REGION Network 13: MB3 Code 3034 - Rotazione Ribalta -AX_POS
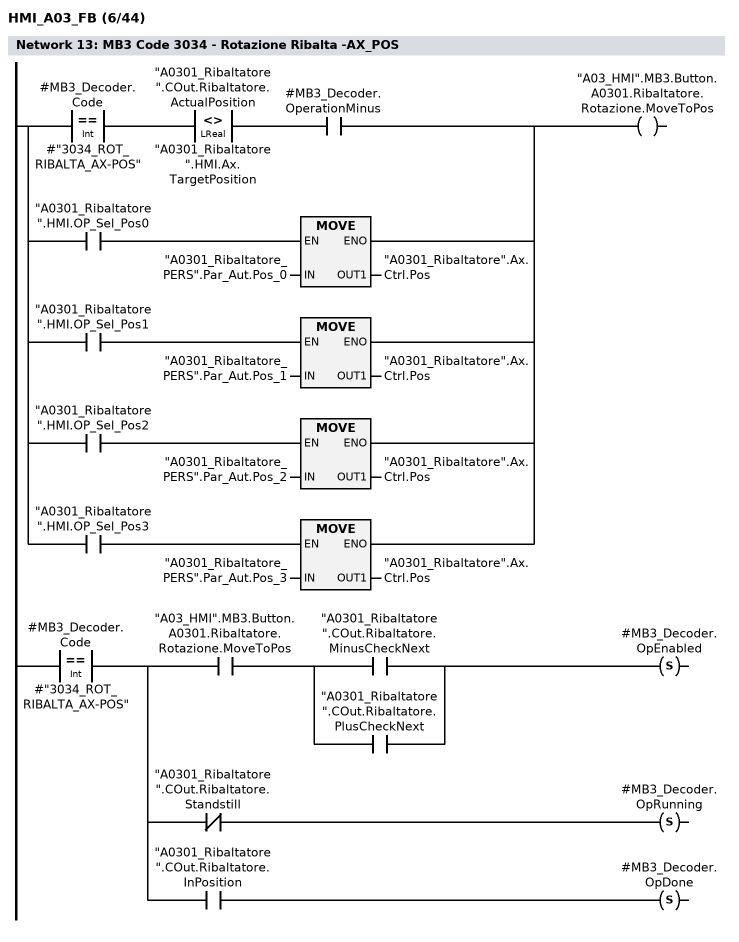
   RUNG wire#powerrail
      { S7_Templates := "SrcType := Int" } EQ_Contact(in1 := #MB3_Decoder.Code, in2 := #"3034_ROT_RIBALTA_AX-POS")
      { S7_Templates := "SrcType := LReal" } NE_Contact(in1 := "A0301_Ribaltatore".COut.Ribaltatore.ActualPosition, in2 := "A0301_Ribaltatore".HMI.Ax.TargetPosition)
      Contact( #MB3_Decoder.OperationMinus )
      wire#w1
      Coil( "A03_HMI".MB3.Button.A0301.Ribaltatore.Rotazione.MoveToPos )
   END_RUNG
   RUNG wire#powerrail
      Contact( "A0301_Ribaltatore".HMI.OP_Sel_Pos0 )
      Move(in := "A0301_Ribaltatore_PERS".Par_Aut.Pos_0, out1 => "A0301_Ribaltatore".Ax.Ctrl.Pos)
   END_RUNG wire#w1
   RUNG wire#powerrail
      Contact( "A0301_Ribaltatore".HMI.OP_Sel_Pos1 )
      Move(in := "A0301_Ribaltatore_PERS".Par_Aut.Pos_1, out1 => "A0301_Ribaltatore".Ax.Ctrl.Pos)
   END_RUNG wire#w1
   RUNG wire#powerrail
      Contact( "A0301_Ribaltatore".HMI.OP_Sel_Pos2 )
      Move(in := "A0301_Ribaltatore_PERS".Par_Aut.Pos_2, out1 => "A0301_Ribaltatore".Ax.Ctrl.Pos)
   END_RUNG wire#w1
   RUNG wire#powerrail
      Contact( "A0301_Ribaltatore".HMI.OP_Sel_Pos3 )
      Move(in := "A0301_Ribaltatore_PERS".Par_Aut.Pos_3, out1 => "A0301_Ribaltatore".Ax.Ctrl.Pos)
   END_RUNG wire#w1
   RUNG wire#powerrail
      { S7_Templates := "SrcType := Int" } EQ_Contact(in1 := #MB3_Decoder.Code, in2 := #"3034_ROT_RIBALTA_AX-POS")
      wire#w2
      Contact( "A03_HMI".MB3.Button.A0301.Ribaltatore.Rotazione.MoveToPos )
      wire#w3
      Contact( "A0301_Ribaltatore".COut.Ribaltatore.MinusCheckNext )
      wire#w4
      S_Coil( #MB3_Decoder.OpEnabled )
   END_RUNG
   RUNG wire#w3
      Contact( "A0301_Ribaltatore".COut.Ribaltatore.PlusCheckNext )
   END_RUNG wire#w4
   RUNG wire#w2
      I_Contact( "A0301_Ribaltatore".COut.Ribaltatore.Standstill )
      S_Coil( #MB3_Decoder.OpRunning )
   END_RUNG
   RUNG wire#w2
      Contact( "A0301_Ribaltatore".COut.Ribaltatore.InPosition )
      S_Coil( #MB3_Decoder.OpDone )
   END_RUNG
   // the same network as SCL:
   IF "A0301_Ribaltatore".HMI.OP_Sel_Pos0 THEN
       "A0301_Ribaltatore".Ax.Ctrl.Pos := "A0301_Ribaltatore_PERS".Par_Aut.Pos_0;
   END_IF;
   IF "A0301_Ribaltatore".HMI.OP_Sel_Pos1 THEN
       "A0301_Ribaltatore".Ax.Ctrl.Pos := "A0301_Ribaltatore_PERS".Par_Aut.Pos_1;
   END_IF;
   IF "A0301_Ribaltatore".HMI.OP_Sel_Pos2 THEN
       "A0301_Ribaltatore".Ax.Ctrl.Pos := "A0301_Ribaltatore_PERS".Par_Aut.Pos_2;
   END_IF;
   IF "A0301_Ribaltatore".HMI.OP_Sel_Pos3 THEN
       "A0301_Ribaltatore".Ax.Ctrl.Pos := "A0301_Ribaltatore_PERS".Par_Aut.Pos_3;
   END_IF;
   "A03_HMI".MB3.Button.A0301.Ribaltatore.Rotazione.MoveToPos := ((#MB3_Decoder.Code = #"3034_ROT_RIBALTA_AX-POS") AND ("A0301_Ribaltatore".COut.Ribaltatore.ActualPosition <> "A0301_Ribaltatore".HMI.Ax.TargetPosition) AND #MB3_Decoder.OperationMinus) OR "A0301_Ribaltatore".HMI.OP_Sel_Pos0 OR "A0301_Ribaltatore".HMI.OP_Sel_Pos1 OR "A0301_Ribaltatore".HMI.OP_Sel_Pos2 OR "A0301_Ribaltatore".HMI.OP_Sel_Pos3;
   #_w1 := #MB3_Decoder.Code = #"3034_ROT_RIBALTA_AX-POS";
   IF #_w1 AND "A03_HMI".MB3.Button.A0301.Ribaltatore.Rotazione.MoveToPos AND ("A0301_Ribaltatore".COut.Ribaltatore.MinusCheckNext OR "A0301_Ribaltatore".COut.Ribaltatore.PlusCheckNext) THEN
       #MB3_Decoder.OpEnabled := TRUE;
   END_IF;
   IF #_w1 AND NOT "A0301_Ribaltatore".COut.Ribaltatore.Standstill THEN
       #MB3_Decoder.OpRunning := TRUE;
   END_IF;
   IF #_w1 AND "A0301_Ribaltatore".COut.Ribaltatore.InPosition THEN #MB3_Decoder.OpDone := TRUE; END_IF;
END_REGION

REGION Network 14: MB3 Code 6008 - Rotazione Ribalta - OP POS0
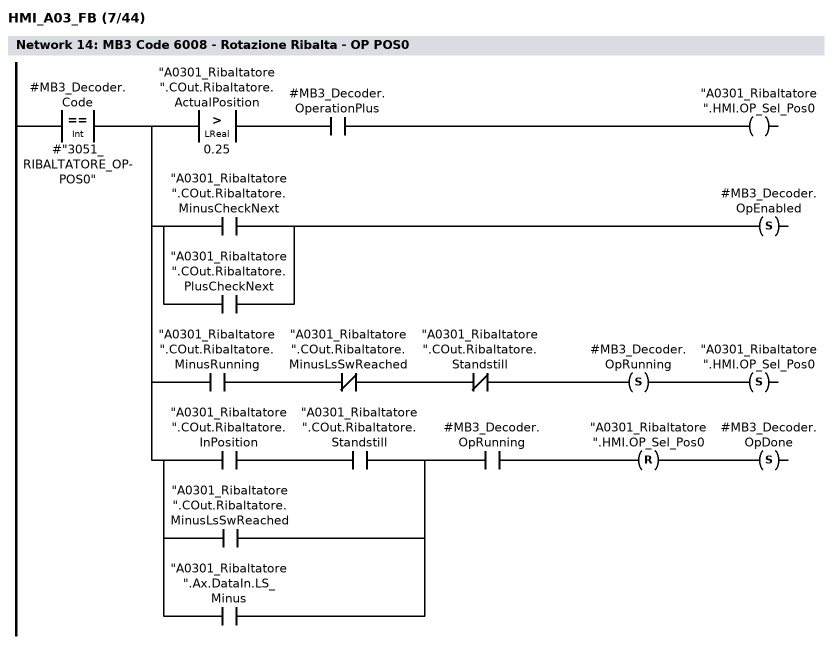
   RUNG wire#powerrail
      { S7_Templates := "SrcType := Int" } EQ_Contact(in1 := #MB3_Decoder.Code, in2 := #"3051_RIBALTATORE_OP-POS0")
      wire#w1
      { S7_Templates := "SrcType := LReal" } GT_Contact(in1 := "A0301_Ribaltatore".COut.Ribaltatore.ActualPosition, in2 := 0.25)
      Contact( #MB3_Decoder.OperationPlus )
      Coil( "A0301_Ribaltatore".HMI.OP_Sel_Pos0 )
   END_RUNG
   RUNG wire#w1
      Contact( "A0301_Ribaltatore".COut.Ribaltatore.MinusCheckNext )
      wire#w2
      S_Coil( #MB3_Decoder.OpEnabled )
   END_RUNG
   RUNG wire#w1
      Contact( "A0301_Ribaltatore".COut.Ribaltatore.PlusCheckNext )
   END_RUNG wire#w2
   RUNG wire#w1
      Contact( "A0301_Ribaltatore".COut.Ribaltatore.MinusRunning )
      I_Contact( "A0301_Ribaltatore".COut.Ribaltatore.MinusLsSwReached )
      I_Contact( "A0301_Ribaltatore".COut.Ribaltatore.Standstill )
      S_Coil( #MB3_Decoder.OpRunning )
      S_Coil( "A0301_Ribaltatore".HMI.OP_Sel_Pos0 )
   END_RUNG
   RUNG wire#w1
      Contact( "A0301_Ribaltatore".COut.Ribaltatore.InPosition )
      Contact( "A0301_Ribaltatore".COut.Ribaltatore.Standstill )
      wire#w3
      Contact( #MB3_Decoder.OpRunning )
      R_Coil( "A0301_Ribaltatore".HMI.OP_Sel_Pos0 )
      S_Coil( #MB3_Decoder.OpDone )
   END_RUNG
   RUNG wire#w1
      Contact( "A0301_Ribaltatore".COut.Ribaltatore.MinusLsSwReached )
   END_RUNG wire#w3
   RUNG wire#w1
      Contact( "A0301_Ribaltatore".Ax.DataIn.LS_Minus )
   END_RUNG wire#w3
   // the same network as SCL:
   #_w1 := #MB3_Decoder.Code = #"3051_RIBALTATORE_OP-POS0";
   "A0301_Ribaltatore".HMI.OP_Sel_Pos0 := #_w1 AND ("A0301_Ribaltatore".COut.Ribaltatore.ActualPosition > 0.25) AND #MB3_Decoder.OperationPlus;
   IF #_w1 AND ("A0301_Ribaltatore".COut.Ribaltatore.MinusCheckNext OR "A0301_Ribaltatore".COut.Ribaltatore.PlusCheckNext) THEN
       #MB3_Decoder.OpEnabled := TRUE;
   END_IF;
   IF #_w1 AND "A0301_Ribaltatore".COut.Ribaltatore.MinusRunning AND NOT "A0301_Ribaltatore".COut.Ribaltatore.MinusLsSwReached AND NOT "A0301_Ribaltatore".COut.Ribaltatore.Standstill THEN
       #MB3_Decoder.OpRunning := TRUE;
       "A0301_Ribaltatore".HMI.OP_Sel_Pos0 := TRUE;
   END_IF;
   IF #_w1 AND (("A0301_Ribaltatore".COut.Ribaltatore.InPosition AND "A0301_Ribaltatore".COut.Ribaltatore.Standstill) OR "A0301_Ribaltatore".COut.Ribaltatore.MinusLsSwReached OR "A0301_Ribaltatore".Ax.DataIn.LS_Minus) AND #MB3_Decoder.OpRunning THEN
       "A0301_Ribaltatore".HMI.OP_Sel_Pos0 := FALSE;
       #MB3_Decoder.OpDone := TRUE;
   END_IF;
END_REGION

REGION Network 15: MB3 Code 6009 - Rotazione Ribalta - OP POS1
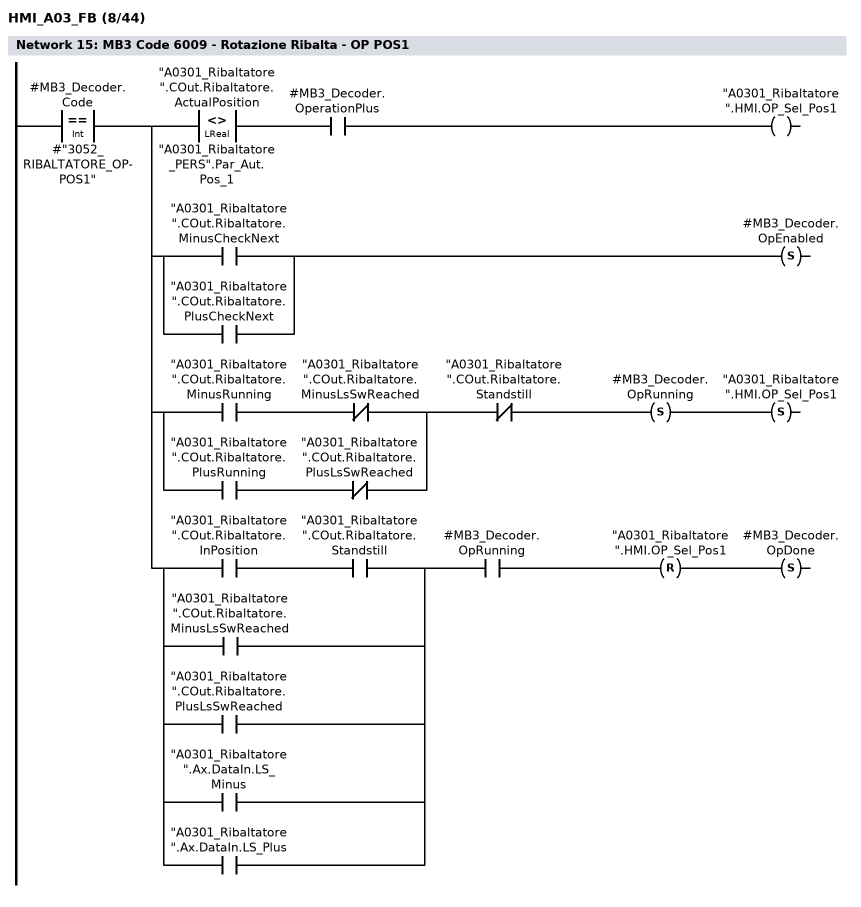
   RUNG wire#powerrail
      { S7_Templates := "SrcType := Int" } EQ_Contact(in1 := #MB3_Decoder.Code, in2 := #"3052_RIBALTATORE_OP-POS1")
      wire#w1
      { S7_Templates := "SrcType := LReal" } NE_Contact(in1 := "A0301_Ribaltatore".COut.Ribaltatore.ActualPosition, in2 := "A0301_Ribaltatore_PERS".Par_Aut.Pos_1)
      Contact( #MB3_Decoder.OperationPlus )
      Coil( "A0301_Ribaltatore".HMI.OP_Sel_Pos1 )
   END_RUNG
   RUNG wire#w1
      Contact( "A0301_Ribaltatore".COut.Ribaltatore.MinusCheckNext )
      wire#w2
      S_Coil( #MB3_Decoder.OpEnabled )
   END_RUNG
   RUNG wire#w1
      Contact( "A0301_Ribaltatore".COut.Ribaltatore.PlusCheckNext )
   END_RUNG wire#w2
   RUNG wire#w1
      Contact( "A0301_Ribaltatore".COut.Ribaltatore.MinusRunning )
      I_Contact( "A0301_Ribaltatore".COut.Ribaltatore.MinusLsSwReached )
      wire#w3
      I_Contact( "A0301_Ribaltatore".COut.Ribaltatore.Standstill )
      S_Coil( #MB3_Decoder.OpRunning )
      S_Coil( "A0301_Ribaltatore".HMI.OP_Sel_Pos1 )
   END_RUNG
   RUNG wire#w1
      Contact( "A0301_Ribaltatore".COut.Ribaltatore.PlusRunning )
      I_Contact( "A0301_Ribaltatore".COut.Ribaltatore.PlusLsSwReached )
   END_RUNG wire#w3
   RUNG wire#w1
      Contact( "A0301_Ribaltatore".COut.Ribaltatore.InPosition )
      Contact( "A0301_Ribaltatore".COut.Ribaltatore.Standstill )
      wire#w4
      Contact( #MB3_Decoder.OpRunning )
      R_Coil( "A0301_Ribaltatore".HMI.OP_Sel_Pos1 )
      S_Coil( #MB3_Decoder.OpDone )
   END_RUNG
   RUNG wire#w1
      Contact( "A0301_Ribaltatore".COut.Ribaltatore.MinusLsSwReached )
   END_RUNG wire#w4
   RUNG wire#w1
      Contact( "A0301_Ribaltatore".COut.Ribaltatore.PlusLsSwReached )
   END_RUNG wire#w4
   RUNG wire#w1
      Contact( "A0301_Ribaltatore".Ax.DataIn.LS_Minus )
   END_RUNG wire#w4
   RUNG wire#w1
      Contact( "A0301_Ribaltatore".Ax.DataIn.LS_Plus )
   END_RUNG wire#w4
   // the same network as SCL:
   #_w1 := #MB3_Decoder.Code = #"3052_RIBALTATORE_OP-POS1";
   "A0301_Ribaltatore".HMI.OP_Sel_Pos1 := #_w1 AND ("A0301_Ribaltatore".COut.Ribaltatore.ActualPosition <> "A0301_Ribaltatore_PERS".Par_Aut.Pos_1) AND #MB3_Decoder.OperationPlus;
   IF #_w1 AND ("A0301_Ribaltatore".COut.Ribaltatore.MinusCheckNext OR "A0301_Ribaltatore".COut.Ribaltatore.PlusCheckNext) THEN
       #MB3_Decoder.OpEnabled := TRUE;
   END_IF;
   IF #_w1 AND (("A0301_Ribaltatore".COut.Ribaltatore.MinusRunning AND NOT "A0301_Ribaltatore".COut.Ribaltatore.MinusLsSwReached) OR ("A0301_Ribaltatore".COut.Ribaltatore.PlusRunning AND NOT "A0301_Ribaltatore".COut.Ribaltatore.PlusLsSwReached)) AND NOT "A0301_Ribaltatore".COut.Ribaltatore.Standstill THEN
       #MB3_Decoder.OpRunning := TRUE;
       "A0301_Ribaltatore".HMI.OP_Sel_Pos1 := TRUE;
   END_IF;
   IF #_w1 AND (("A0301_Ribaltatore".COut.Ribaltatore.InPosition AND "A0301_Ribaltatore".COut.Ribaltatore.Standstill) OR "A0301_Ribaltatore".COut.Ribaltatore.MinusLsSwReached OR "A0301_Ribaltatore".COut.Ribaltatore.PlusLsSwReached OR "A0301_Ribaltatore".Ax.DataIn.LS_Minus OR "A0301_Ribaltatore".Ax.DataIn.LS_Plus) AND #MB3_Decoder.OpRunning THEN
       "A0301_Ribaltatore".HMI.OP_Sel_Pos1 := FALSE;
       #MB3_Decoder.OpDone := TRUE;
   END_IF;
END_REGION

REGION Network 16: MB3 Code 6010 - Rotazione Ribalta - OP POS2
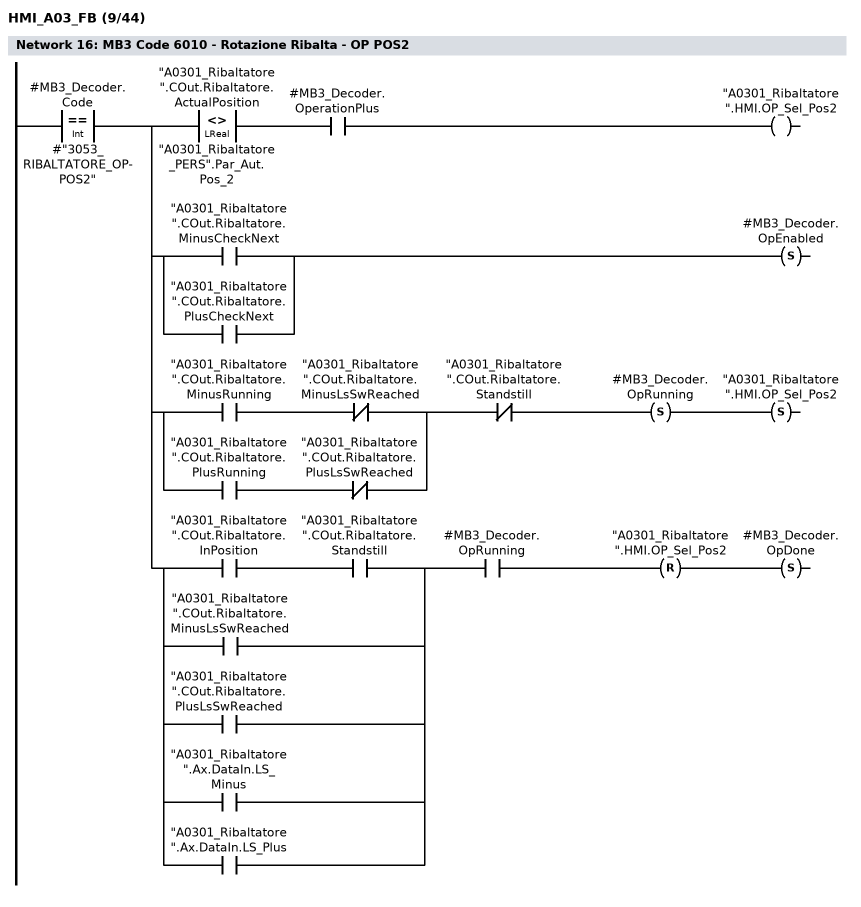
   RUNG wire#powerrail
      { S7_Templates := "SrcType := Int" } EQ_Contact(in1 := #MB3_Decoder.Code, in2 := #"3053_RIBALTATORE_OP-POS2")
      wire#w1
      { S7_Templates := "SrcType := LReal" } NE_Contact(in1 := "A0301_Ribaltatore".COut.Ribaltatore.ActualPosition, in2 := "A0301_Ribaltatore_PERS".Par_Aut.Pos_2)
      Contact( #MB3_Decoder.OperationPlus )
      Coil( "A0301_Ribaltatore".HMI.OP_Sel_Pos2 )
   END_RUNG
   RUNG wire#w1
      Contact( "A0301_Ribaltatore".COut.Ribaltatore.MinusCheckNext )
      wire#w2
      S_Coil( #MB3_Decoder.OpEnabled )
   END_RUNG
   RUNG wire#w1
      Contact( "A0301_Ribaltatore".COut.Ribaltatore.PlusCheckNext )
   END_RUNG wire#w2
   RUNG wire#w1
      Contact( "A0301_Ribaltatore".COut.Ribaltatore.MinusRunning )
      I_Contact( "A0301_Ribaltatore".COut.Ribaltatore.MinusLsSwReached )
      wire#w3
      I_Contact( "A0301_Ribaltatore".COut.Ribaltatore.Standstill )
      S_Coil( #MB3_Decoder.OpRunning )
      S_Coil( "A0301_Ribaltatore".HMI.OP_Sel_Pos2 )
   END_RUNG
   RUNG wire#w1
      Contact( "A0301_Ribaltatore".COut.Ribaltatore.PlusRunning )
      I_Contact( "A0301_Ribaltatore".COut.Ribaltatore.PlusLsSwReached )
   END_RUNG wire#w3
   RUNG wire#w1
      Contact( "A0301_Ribaltatore".COut.Ribaltatore.InPosition )
      Contact( "A0301_Ribaltatore".COut.Ribaltatore.Standstill )
      wire#w4
      Contact( #MB3_Decoder.OpRunning )
      R_Coil( "A0301_Ribaltatore".HMI.OP_Sel_Pos2 )
      S_Coil( #MB3_Decoder.OpDone )
   END_RUNG
   RUNG wire#w1
      Contact( "A0301_Ribaltatore".COut.Ribaltatore.MinusLsSwReached )
   END_RUNG wire#w4
   RUNG wire#w1
      Contact( "A0301_Ribaltatore".COut.Ribaltatore.PlusLsSwReached )
   END_RUNG wire#w4
   RUNG wire#w1
      Contact( "A0301_Ribaltatore".Ax.DataIn.LS_Minus )
   END_RUNG wire#w4
   RUNG wire#w1
      Contact( "A0301_Ribaltatore".Ax.DataIn.LS_Plus )
   END_RUNG wire#w4
   // the same network as SCL:
   #_w1 := #MB3_Decoder.Code = #"3053_RIBALTATORE_OP-POS2";
   "A0301_Ribaltatore".HMI.OP_Sel_Pos2 := #_w1 AND ("A0301_Ribaltatore".COut.Ribaltatore.ActualPosition <> "A0301_Ribaltatore_PERS".Par_Aut.Pos_2) AND #MB3_Decoder.OperationPlus;
   IF #_w1 AND ("A0301_Ribaltatore".COut.Ribaltatore.MinusCheckNext OR "A0301_Ribaltatore".COut.Ribaltatore.PlusCheckNext) THEN
       #MB3_Decoder.OpEnabled := TRUE;
   END_IF;
   IF #_w1 AND (("A0301_Ribaltatore".COut.Ribaltatore.MinusRunning AND NOT "A0301_Ribaltatore".COut.Ribaltatore.MinusLsSwReached) OR ("A0301_Ribaltatore".COut.Ribaltatore.PlusRunning AND NOT "A0301_Ribaltatore".COut.Ribaltatore.PlusLsSwReached)) AND NOT "A0301_Ribaltatore".COut.Ribaltatore.Standstill THEN
       #MB3_Decoder.OpRunning := TRUE;
       "A0301_Ribaltatore".HMI.OP_Sel_Pos2 := TRUE;
   END_IF;
   IF #_w1 AND (("A0301_Ribaltatore".COut.Ribaltatore.InPosition AND "A0301_Ribaltatore".COut.Ribaltatore.Standstill) OR "A0301_Ribaltatore".COut.Ribaltatore.MinusLsSwReached OR "A0301_Ribaltatore".COut.Ribaltatore.PlusLsSwReached OR "A0301_Ribaltatore".Ax.DataIn.LS_Minus OR "A0301_Ribaltatore".Ax.DataIn.LS_Plus) AND #MB3_Decoder.OpRunning THEN
       "A0301_Ribaltatore".HMI.OP_Sel_Pos2 := FALSE;
       #MB3_Decoder.OpDone := TRUE;
   END_IF;
END_REGION

REGION Network 17: MB3 Code 6011 - Rotazione Ribalta - OP POS3
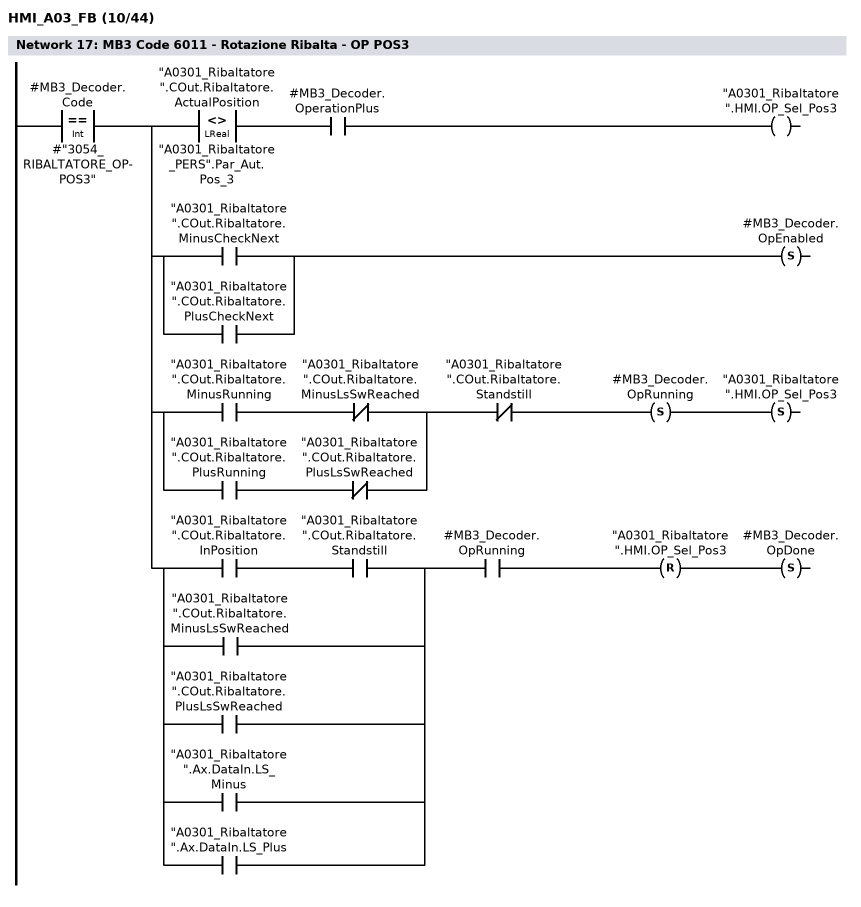
   RUNG wire#powerrail
      { S7_Templates := "SrcType := Int" } EQ_Contact(in1 := #MB3_Decoder.Code, in2 := #"3054_RIBALTATORE_OP-POS3")
      wire#w1
      { S7_Templates := "SrcType := LReal" } NE_Contact(in1 := "A0301_Ribaltatore".COut.Ribaltatore.ActualPosition, in2 := "A0301_Ribaltatore_PERS".Par_Aut.Pos_3)
      Contact( #MB3_Decoder.OperationPlus )
      Coil( "A0301_Ribaltatore".HMI.OP_Sel_Pos3 )
   END_RUNG
   RUNG wire#w1
      Contact( "A0301_Ribaltatore".COut.Ribaltatore.MinusCheckNext )
      wire#w2
      S_Coil( #MB3_Decoder.OpEnabled )
   END_RUNG
   RUNG wire#w1
      Contact( "A0301_Ribaltatore".COut.Ribaltatore.PlusCheckNext )
   END_RUNG wire#w2
   RUNG wire#w1
      Contact( "A0301_Ribaltatore".COut.Ribaltatore.MinusRunning )
      I_Contact( "A0301_Ribaltatore".COut.Ribaltatore.MinusLsSwReached )
      wire#w3
      I_Contact( "A0301_Ribaltatore".COut.Ribaltatore.Standstill )
      S_Coil( #MB3_Decoder.OpRunning )
      S_Coil( "A0301_Ribaltatore".HMI.OP_Sel_Pos3 )
   END_RUNG
   RUNG wire#w1
      Contact( "A0301_Ribaltatore".COut.Ribaltatore.PlusRunning )
      I_Contact( "A0301_Ribaltatore".COut.Ribaltatore.PlusLsSwReached )
   END_RUNG wire#w3
   RUNG wire#w1
      Contact( "A0301_Ribaltatore".COut.Ribaltatore.InPosition )
      Contact( "A0301_Ribaltatore".COut.Ribaltatore.Standstill )
      wire#w4
      Contact( #MB3_Decoder.OpRunning )
      R_Coil( "A0301_Ribaltatore".HMI.OP_Sel_Pos3 )
      S_Coil( #MB3_Decoder.OpDone )
   END_RUNG
   RUNG wire#w1
      Contact( "A0301_Ribaltatore".COut.Ribaltatore.MinusLsSwReached )
   END_RUNG wire#w4
   RUNG wire#w1
      Contact( "A0301_Ribaltatore".COut.Ribaltatore.PlusLsSwReached )
   END_RUNG wire#w4
   RUNG wire#w1
      Contact( "A0301_Ribaltatore".Ax.DataIn.LS_Minus )
   END_RUNG wire#w4
   RUNG wire#w1
      Contact( "A0301_Ribaltatore".Ax.DataIn.LS_Plus )
   END_RUNG wire#w4
   // the same network as SCL:
   #_w1 := #MB3_Decoder.Code = #"3054_RIBALTATORE_OP-POS3";
   "A0301_Ribaltatore".HMI.OP_Sel_Pos3 := #_w1 AND ("A0301_Ribaltatore".COut.Ribaltatore.ActualPosition <> "A0301_Ribaltatore_PERS".Par_Aut.Pos_3) AND #MB3_Decoder.OperationPlus;
   IF #_w1 AND ("A0301_Ribaltatore".COut.Ribaltatore.MinusCheckNext OR "A0301_Ribaltatore".COut.Ribaltatore.PlusCheckNext) THEN
       #MB3_Decoder.OpEnabled := TRUE;
   END_IF;
   IF #_w1 AND (("A0301_Ribaltatore".COut.Ribaltatore.MinusRunning AND NOT "A0301_Ribaltatore".COut.Ribaltatore.MinusLsSwReached) OR ("A0301_Ribaltatore".COut.Ribaltatore.PlusRunning AND NOT "A0301_Ribaltatore".COut.Ribaltatore.PlusLsSwReached)) AND NOT "A0301_Ribaltatore".COut.Ribaltatore.Standstill THEN
       #MB3_Decoder.OpRunning := TRUE;
       "A0301_Ribaltatore".HMI.OP_Sel_Pos3 := TRUE;
   END_IF;
   IF #_w1 AND (("A0301_Ribaltatore".COut.Ribaltatore.InPosition AND "A0301_Ribaltatore".COut.Ribaltatore.Standstill) OR "A0301_Ribaltatore".COut.Ribaltatore.MinusLsSwReached OR "A0301_Ribaltatore".COut.Ribaltatore.PlusLsSwReached OR "A0301_Ribaltatore".Ax.DataIn.LS_Minus OR "A0301_Ribaltatore".Ax.DataIn.LS_Plus) AND #MB3_Decoder.OpRunning THEN
       "A0301_Ribaltatore".HMI.OP_Sel_Pos3 := FALSE;
       #MB3_Decoder.OpDone := TRUE;
   END_IF;
END_REGION

REGION Network 18: MB3 Code 3041 - Fermi P4
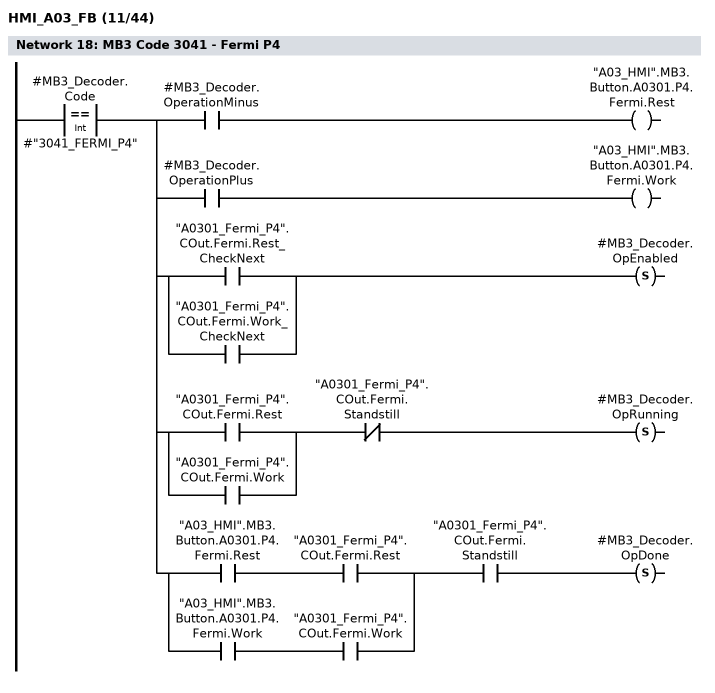
   RUNG wire#powerrail
      { S7_Templates := "SrcType := Int" } EQ_Contact(in1 := #MB3_Decoder.Code, in2 := #"3041_FERMI_P4")
      wire#w1
      Contact( #MB3_Decoder.OperationMinus )
      Coil( "A03_HMI".MB3.Button.A0301.P4.Fermi.Rest )
   END_RUNG
   RUNG wire#w1
      Contact( #MB3_Decoder.OperationPlus )
      Coil( "A03_HMI".MB3.Button.A0301.P4.Fermi.Work )
   END_RUNG
   RUNG wire#w1
      Contact( "A0301_Fermi_P4".COut.Fermi.Rest_CheckNext )
      wire#w2
      S_Coil( #MB3_Decoder.OpEnabled )
   END_RUNG
   RUNG wire#w1
      Contact( "A0301_Fermi_P4".COut.Fermi.Work_CheckNext )
   END_RUNG wire#w2
   RUNG wire#w1
      Contact( "A0301_Fermi_P4".COut.Fermi.Rest )
      wire#w3
      I_Contact( "A0301_Fermi_P4".COut.Fermi.Standstill )
      S_Coil( #MB3_Decoder.OpRunning )
   END_RUNG
   RUNG wire#w1
      Contact( "A0301_Fermi_P4".COut.Fermi.Work )
   END_RUNG wire#w3
   RUNG wire#w1
      Contact( "A03_HMI".MB3.Button.A0301.P4.Fermi.Rest )
      Contact( "A0301_Fermi_P4".COut.Fermi.Rest )
      wire#w4
      Contact( "A0301_Fermi_P4".COut.Fermi.Standstill )
      S_Coil( #MB3_Decoder.OpDone )
   END_RUNG
   RUNG wire#w1
      Contact( "A03_HMI".MB3.Button.A0301.P4.Fermi.Work )
      Contact( "A0301_Fermi_P4".COut.Fermi.Work )
   END_RUNG wire#w4
   // the same network as SCL:
   #_w1 := #MB3_Decoder.Code = #"3041_FERMI_P4";
   "A03_HMI".MB3.Button.A0301.P4.Fermi.Rest := #_w1 AND #MB3_Decoder.OperationMinus;
   "A03_HMI".MB3.Button.A0301.P4.Fermi.Work := #_w1 AND #MB3_Decoder.OperationPlus;
   IF #_w1 AND ("A0301_Fermi_P4".COut.Fermi.Rest_CheckNext OR "A0301_Fermi_P4".COut.Fermi.Work_CheckNext) THEN
       #MB3_Decoder.OpEnabled := TRUE;
   END_IF;
   IF #_w1 AND ("A0301_Fermi_P4".COut.Fermi.Rest OR "A0301_Fermi_P4".COut.Fermi.Work) AND NOT "A0301_Fermi_P4".COut.Fermi.Standstill THEN
       #MB3_Decoder.OpRunning := TRUE;
   END_IF;
   IF #_w1 AND (("A03_HMI".MB3.Button.A0301.P4.Fermi.Rest AND "A0301_Fermi_P4".COut.Fermi.Rest) OR ("A03_HMI".MB3.Button.A0301.P4.Fermi.Work AND "A0301_Fermi_P4".COut.Fermi.Work)) AND "A0301_Fermi_P4".COut.Fermi.Standstill THEN
       #MB3_Decoder.OpDone := TRUE;
   END_IF;
END_REGION

REGION Network 19: MB3 Code 3042 - P5 - Spintore Laterale-Vrt
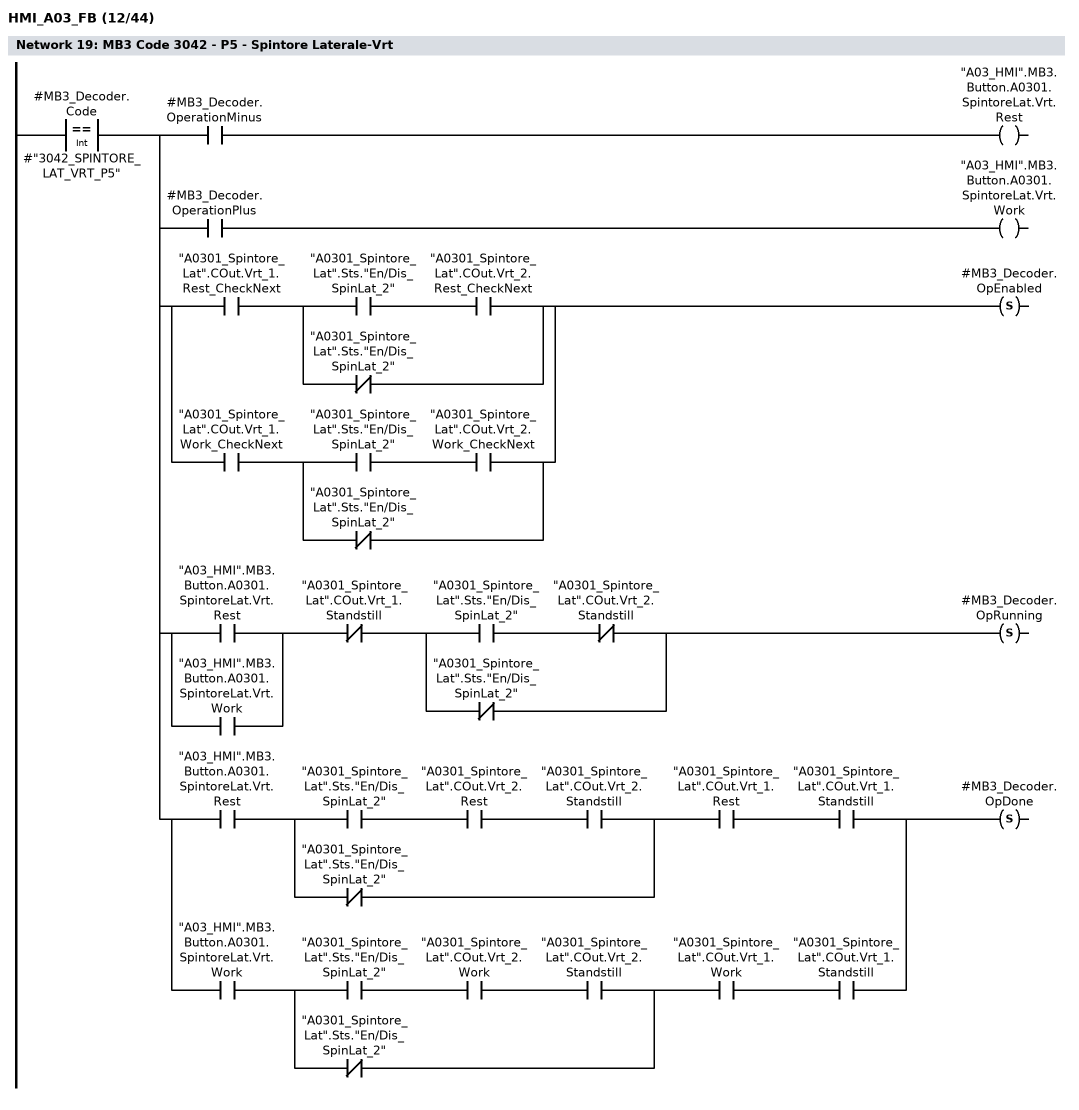
   RUNG wire#powerrail
      { S7_Templates := "SrcType := Int" } EQ_Contact(in1 := #MB3_Decoder.Code, in2 := #"3042_SPINTORE_LAT_VRT_P5")
      wire#w1
      Contact( #MB3_Decoder.OperationMinus )
      Coil( "A03_HMI".MB3.Button.A0301.SpintoreLat.Vrt.Rest )
   END_RUNG
   RUNG wire#w1
      Contact( #MB3_Decoder.OperationPlus )
      Coil( "A03_HMI".MB3.Button.A0301.SpintoreLat.Vrt.Work )
   END_RUNG
   RUNG wire#w1
      Contact( "A0301_Spintore_Lat".COut.Vrt_1.Rest_CheckNext )
      wire#w2
      Contact( "A0301_Spintore_Lat".Sts."En/Dis_SpinLat_2" )
      Contact( "A0301_Spintore_Lat".COut.Vrt_2.Rest_CheckNext )
      wire#w3
      S_Coil( #MB3_Decoder.OpEnabled )
   END_RUNG
   RUNG wire#w2
      I_Contact( "A0301_Spintore_Lat".Sts."En/Dis_SpinLat_2" )
   END_RUNG wire#w3
   RUNG wire#w1
      Contact( "A0301_Spintore_Lat".COut.Vrt_1.Work_CheckNext )
      wire#w4
      Contact( "A0301_Spintore_Lat".Sts."En/Dis_SpinLat_2" )
      Contact( "A0301_Spintore_Lat".COut.Vrt_2.Work_CheckNext )
   END_RUNG wire#w3
   RUNG wire#w4
      I_Contact( "A0301_Spintore_Lat".Sts."En/Dis_SpinLat_2" )
   END_RUNG wire#w3
   RUNG wire#w1
      Contact( "A03_HMI".MB3.Button.A0301.SpintoreLat.Vrt.Rest )
      wire#w5
      I_Contact( "A0301_Spintore_Lat".COut.Vrt_1.Standstill )
      wire#w6
      Contact( "A0301_Spintore_Lat".Sts."En/Dis_SpinLat_2" )
      I_Contact( "A0301_Spintore_Lat".COut.Vrt_2.Standstill )
      wire#w7
      S_Coil( #MB3_Decoder.OpRunning )
   END_RUNG
   RUNG wire#w1
      Contact( "A03_HMI".MB3.Button.A0301.SpintoreLat.Vrt.Work )
   END_RUNG wire#w5
   RUNG wire#w6
      I_Contact( "A0301_Spintore_Lat".Sts."En/Dis_SpinLat_2" )
   END_RUNG wire#w7
   RUNG wire#w1
      Contact( "A03_HMI".MB3.Button.A0301.SpintoreLat.Vrt.Rest )
      wire#w8
      Contact( "A0301_Spintore_Lat".Sts."En/Dis_SpinLat_2" )
      Contact( "A0301_Spintore_Lat".COut.Vrt_2.Rest )
      Contact( "A0301_Spintore_Lat".COut.Vrt_2.Standstill )
      wire#w9
      Contact( "A0301_Spintore_Lat".COut.Vrt_1.Rest )
      Contact( "A0301_Spintore_Lat".COut.Vrt_1.Standstill )
      wire#w10
      S_Coil( #MB3_Decoder.OpDone )
   END_RUNG
   RUNG wire#w8
      I_Contact( "A0301_Spintore_Lat".Sts."En/Dis_SpinLat_2" )
   END_RUNG wire#w9
   RUNG wire#w1
      Contact( "A03_HMI".MB3.Button.A0301.SpintoreLat.Vrt.Work )
      wire#w11
      Contact( "A0301_Spintore_Lat".Sts."En/Dis_SpinLat_2" )
      Contact( "A0301_Spintore_Lat".COut.Vrt_2.Work )
      Contact( "A0301_Spintore_Lat".COut.Vrt_2.Standstill )
      wire#w12
      Contact( "A0301_Spintore_Lat".COut.Vrt_1.Work )
      Contact( "A0301_Spintore_Lat".COut.Vrt_1.Standstill )
   END_RUNG wire#w10
   RUNG wire#w11
      I_Contact( "A0301_Spintore_Lat".Sts."En/Dis_SpinLat_2" )
   END_RUNG wire#w12
   // the same network as SCL:
   #_w1 := #MB3_Decoder.Code = #"3042_SPINTORE_LAT_VRT_P5";
   "A03_HMI".MB3.Button.A0301.SpintoreLat.Vrt.Rest := #_w1 AND #MB3_Decoder.OperationMinus;
   "A03_HMI".MB3.Button.A0301.SpintoreLat.Vrt.Work := #_w1 AND #MB3_Decoder.OperationPlus;
   IF #_w1 AND (("A0301_Spintore_Lat".COut.Vrt_1.Rest_CheckNext AND (("A0301_Spintore_Lat".Sts."En/Dis_SpinLat_2" AND "A0301_Spintore_Lat".COut.Vrt_2.Rest_CheckNext) OR NOT "A0301_Spintore_Lat".Sts."En/Dis_SpinLat_2")) OR ("A0301_Spintore_Lat".COut.Vrt_1.Work_CheckNext AND (("A0301_Spintore_Lat".Sts."En/Dis_SpinLat_2" AND "A0301_Spintore_Lat".COut.Vrt_2.Work_CheckNext) OR NOT "A0301_Spintore_Lat".Sts."En/Dis_SpinLat_2"))) THEN
       #MB3_Decoder.OpEnabled := TRUE;
   END_IF;
   IF #_w1 AND ("A03_HMI".MB3.Button.A0301.SpintoreLat.Vrt.Rest OR "A03_HMI".MB3.Button.A0301.SpintoreLat.Vrt.Work) AND NOT "A0301_Spintore_Lat".COut.Vrt_1.Standstill AND (("A0301_Spintore_Lat".Sts."En/Dis_SpinLat_2" AND NOT "A0301_Spintore_Lat".COut.Vrt_2.Standstill) OR NOT "A0301_Spintore_Lat".Sts."En/Dis_SpinLat_2") THEN
       #MB3_Decoder.OpRunning := TRUE;
   END_IF;
   IF #_w1 AND (("A03_HMI".MB3.Button.A0301.SpintoreLat.Vrt.Rest AND (("A0301_Spintore_Lat".Sts."En/Dis_SpinLat_2" AND "A0301_Spintore_Lat".COut.Vrt_2.Rest AND "A0301_Spintore_Lat".COut.Vrt_2.Standstill) OR NOT "A0301_Spintore_Lat".Sts."En/Dis_SpinLat_2") AND "A0301_Spintore_Lat".COut.Vrt_1.Rest AND "A0301_Spintore_Lat".COut.Vrt_1.Standstill) OR ("A03_HMI".MB3.Button.A0301.SpintoreLat.Vrt.Work AND (("A0301_Spintore_Lat".Sts."En/Dis_SpinLat_2" AND "A0301_Spintore_Lat".COut.Vrt_2.Work AND "A0301_Spintore_Lat".COut.Vrt_2.Standstill) OR NOT "A0301_Spintore_Lat".Sts."En/Dis_SpinLat_2") AND "A0301_Spintore_Lat".COut.Vrt_1.Work AND "A0301_Spintore_Lat".COut.Vrt_1.Standstill)) THEN
       #MB3_Decoder.OpDone := TRUE;
   END_IF;
END_REGION

REGION Network 20: MB3 Code 3043 - P5 - Spintore Laterale-Orz
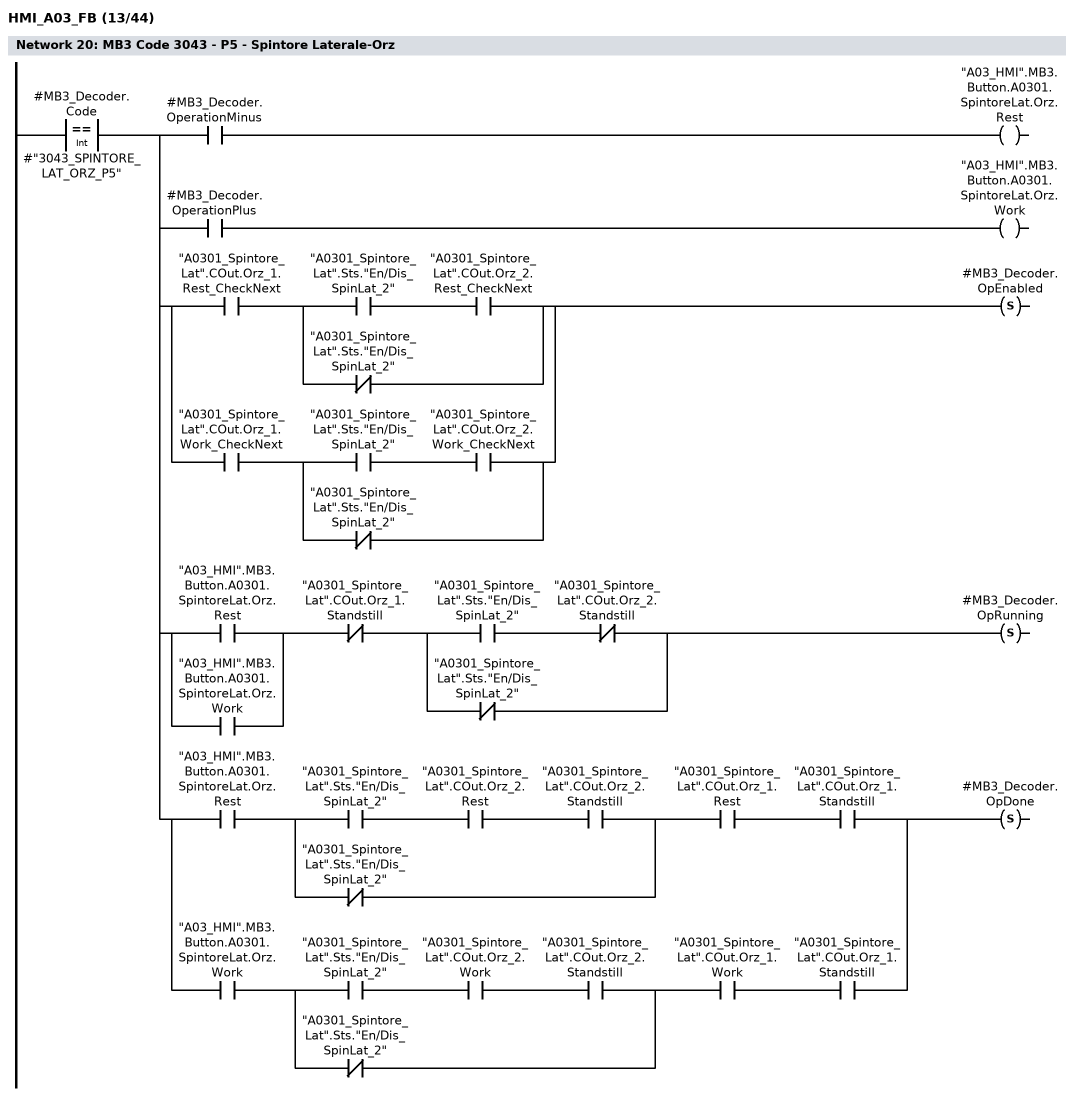
   RUNG wire#powerrail
      { S7_Templates := "SrcType := Int" } EQ_Contact(in1 := #MB3_Decoder.Code, in2 := #"3043_SPINTORE_LAT_ORZ_P5")
      wire#w1
      Contact( #MB3_Decoder.OperationMinus )
      Coil( "A03_HMI".MB3.Button.A0301.SpintoreLat.Orz.Rest )
   END_RUNG
   RUNG wire#w1
      Contact( #MB3_Decoder.OperationPlus )
      Coil( "A03_HMI".MB3.Button.A0301.SpintoreLat.Orz.Work )
   END_RUNG
   RUNG wire#w1
      Contact( "A0301_Spintore_Lat".COut.Orz_1.Rest_CheckNext )
      wire#w2
      Contact( "A0301_Spintore_Lat".Sts."En/Dis_SpinLat_2" )
      Contact( "A0301_Spintore_Lat".COut.Orz_2.Rest_CheckNext )
      wire#w3
      S_Coil( #MB3_Decoder.OpEnabled )
   END_RUNG
   RUNG wire#w2
      I_Contact( "A0301_Spintore_Lat".Sts."En/Dis_SpinLat_2" )
   END_RUNG wire#w3
   RUNG wire#w1
      Contact( "A0301_Spintore_Lat".COut.Orz_1.Work_CheckNext )
      wire#w4
      Contact( "A0301_Spintore_Lat".Sts."En/Dis_SpinLat_2" )
      Contact( "A0301_Spintore_Lat".COut.Orz_2.Work_CheckNext )
   END_RUNG wire#w3
   RUNG wire#w4
      I_Contact( "A0301_Spintore_Lat".Sts."En/Dis_SpinLat_2" )
   END_RUNG wire#w3
   RUNG wire#w1
      Contact( "A03_HMI".MB3.Button.A0301.SpintoreLat.Orz.Rest )
      wire#w5
      I_Contact( "A0301_Spintore_Lat".COut.Orz_1.Standstill )
      wire#w6
      Contact( "A0301_Spintore_Lat".Sts."En/Dis_SpinLat_2" )
      I_Contact( "A0301_Spintore_Lat".COut.Orz_2.Standstill )
      wire#w7
      S_Coil( #MB3_Decoder.OpRunning )
   END_RUNG
   RUNG wire#w1
      Contact( "A03_HMI".MB3.Button.A0301.SpintoreLat.Orz.Work )
   END_RUNG wire#w5
   RUNG wire#w6
      I_Contact( "A0301_Spintore_Lat".Sts."En/Dis_SpinLat_2" )
   END_RUNG wire#w7
   RUNG wire#w1
      Contact( "A03_HMI".MB3.Button.A0301.SpintoreLat.Orz.Rest )
      wire#w8
      Contact( "A0301_Spintore_Lat".Sts."En/Dis_SpinLat_2" )
      Contact( "A0301_Spintore_Lat".COut.Orz_2.Rest )
      Contact( "A0301_Spintore_Lat".COut.Orz_2.Standstill )
      wire#w9
      Contact( "A0301_Spintore_Lat".COut.Orz_1.Rest )
      Contact( "A0301_Spintore_Lat".COut.Orz_1.Standstill )
      wire#w10
      S_Coil( #MB3_Decoder.OpDone )
   END_RUNG
   RUNG wire#w8
      I_Contact( "A0301_Spintore_Lat".Sts."En/Dis_SpinLat_2" )
   END_RUNG wire#w9
   RUNG wire#w1
      Contact( "A03_HMI".MB3.Button.A0301.SpintoreLat.Orz.Work )
      wire#w11
      Contact( "A0301_Spintore_Lat".Sts."En/Dis_SpinLat_2" )
      Contact( "A0301_Spintore_Lat".COut.Orz_2.Work )
      Contact( "A0301_Spintore_Lat".COut.Orz_2.Standstill )
      wire#w12
      Contact( "A0301_Spintore_Lat".COut.Orz_1.Work )
      Contact( "A0301_Spintore_Lat".COut.Orz_1.Standstill )
   END_RUNG wire#w10
   RUNG wire#w11
      I_Contact( "A0301_Spintore_Lat".Sts."En/Dis_SpinLat_2" )
   END_RUNG wire#w12
   // the same network as SCL:
   #_w1 := #MB3_Decoder.Code = #"3043_SPINTORE_LAT_ORZ_P5";
   "A03_HMI".MB3.Button.A0301.SpintoreLat.Orz.Rest := #_w1 AND #MB3_Decoder.OperationMinus;
   "A03_HMI".MB3.Button.A0301.SpintoreLat.Orz.Work := #_w1 AND #MB3_Decoder.OperationPlus;
   IF #_w1 AND (("A0301_Spintore_Lat".COut.Orz_1.Rest_CheckNext AND (("A0301_Spintore_Lat".Sts."En/Dis_SpinLat_2" AND "A0301_Spintore_Lat".COut.Orz_2.Rest_CheckNext) OR NOT "A0301_Spintore_Lat".Sts."En/Dis_SpinLat_2")) OR ("A0301_Spintore_Lat".COut.Orz_1.Work_CheckNext AND (("A0301_Spintore_Lat".Sts."En/Dis_SpinLat_2" AND "A0301_Spintore_Lat".COut.Orz_2.Work_CheckNext) OR NOT "A0301_Spintore_Lat".Sts."En/Dis_SpinLat_2"))) THEN
       #MB3_Decoder.OpEnabled := TRUE;
   END_IF;
   IF #_w1 AND ("A03_HMI".MB3.Button.A0301.SpintoreLat.Orz.Rest OR "A03_HMI".MB3.Button.A0301.SpintoreLat.Orz.Work) AND NOT "A0301_Spintore_Lat".COut.Orz_1.Standstill AND (("A0301_Spintore_Lat".Sts."En/Dis_SpinLat_2" AND NOT "A0301_Spintore_Lat".COut.Orz_2.Standstill) OR NOT "A0301_Spintore_Lat".Sts."En/Dis_SpinLat_2") THEN
       #MB3_Decoder.OpRunning := TRUE;
   END_IF;
   IF #_w1 AND (("A03_HMI".MB3.Button.A0301.SpintoreLat.Orz.Rest AND (("A0301_Spintore_Lat".Sts."En/Dis_SpinLat_2" AND "A0301_Spintore_Lat".COut.Orz_2.Rest AND "A0301_Spintore_Lat".COut.Orz_2.Standstill) OR NOT "A0301_Spintore_Lat".Sts."En/Dis_SpinLat_2") AND "A0301_Spintore_Lat".COut.Orz_1.Rest AND "A0301_Spintore_Lat".COut.Orz_1.Standstill) OR ("A03_HMI".MB3.Button.A0301.SpintoreLat.Orz.Work AND (("A0301_Spintore_Lat".Sts."En/Dis_SpinLat_2" AND "A0301_Spintore_Lat".COut.Orz_2.Work AND "A0301_Spintore_Lat".COut.Orz_2.Standstill) OR NOT "A0301_Spintore_Lat".Sts."En/Dis_SpinLat_2") AND "A0301_Spintore_Lat".COut.Orz_1.Work AND "A0301_Spintore_Lat".COut.Orz_1.Standstill)) THEN
       #MB3_Decoder.OpDone := TRUE;
   END_IF;
END_REGION

REGION Network 21: MB3 Code 3045 - P5 - Spintore Laterale-OP
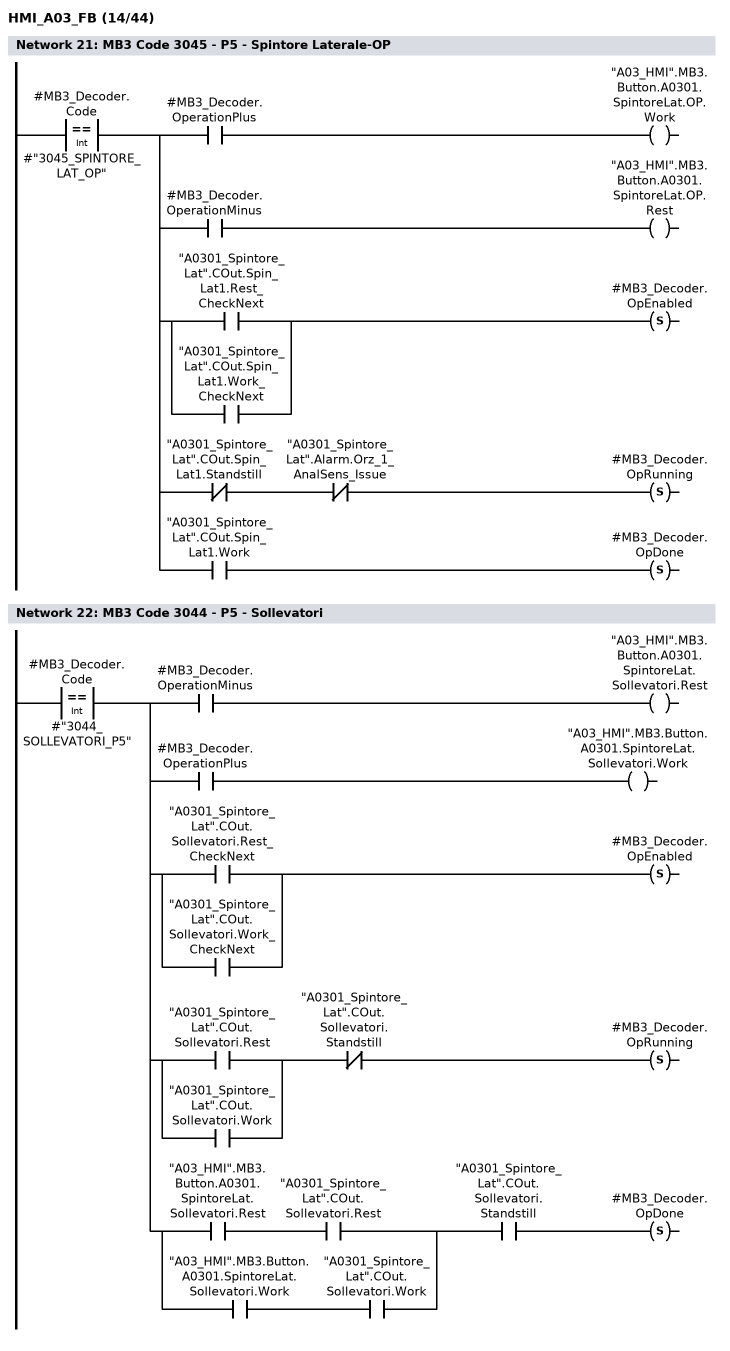
   RUNG wire#powerrail
      { S7_Templates := "SrcType := Int" } EQ_Contact(in1 := #MB3_Decoder.Code, in2 := #"3045_SPINTORE_LAT_OP")
      wire#w1
      Contact( #MB3_Decoder.OperationPlus )
      Coil( "A03_HMI".MB3.Button.A0301.SpintoreLat.OP.Work )
   END_RUNG
   RUNG wire#w1
      Contact( #MB3_Decoder.OperationMinus )
      Coil( "A03_HMI".MB3.Button.A0301.SpintoreLat.OP.Rest )
   END_RUNG
   RUNG wire#w1
      Contact( "A0301_Spintore_Lat".COut.Spin_Lat1.Rest_CheckNext )
      wire#w2
      S_Coil( #MB3_Decoder.OpEnabled )
   END_RUNG
   RUNG wire#w1
      Contact( "A0301_Spintore_Lat".COut.Spin_Lat1.Work_CheckNext )
   END_RUNG wire#w2
   RUNG wire#w1
      I_Contact( "A0301_Spintore_Lat".COut.Spin_Lat1.Standstill )
      I_Contact( "A0301_Spintore_Lat".Alarm.Orz_1_AnalSens_Issue )
      S_Coil( #MB3_Decoder.OpRunning )
   END_RUNG
   RUNG wire#w1
      Contact( "A0301_Spintore_Lat".COut.Spin_Lat1.Work )
      S_Coil( #MB3_Decoder.OpDone )
   END_RUNG
   // the same network as SCL:
   #_w1 := #MB3_Decoder.Code = #"3045_SPINTORE_LAT_OP";
   "A03_HMI".MB3.Button.A0301.SpintoreLat.OP.Work := #_w1 AND #MB3_Decoder.OperationPlus;
   "A03_HMI".MB3.Button.A0301.SpintoreLat.OP.Rest := #_w1 AND #MB3_Decoder.OperationMinus;
   IF #_w1 AND ("A0301_Spintore_Lat".COut.Spin_Lat1.Rest_CheckNext OR "A0301_Spintore_Lat".COut.Spin_Lat1.Work_CheckNext) THEN
       #MB3_Decoder.OpEnabled := TRUE;
   END_IF;
   IF #_w1 AND NOT "A0301_Spintore_Lat".COut.Spin_Lat1.Standstill AND NOT "A0301_Spintore_Lat".Alarm.Orz_1_AnalSens_Issue THEN
       #MB3_Decoder.OpRunning := TRUE;
   END_IF;
   IF #_w1 AND "A0301_Spintore_Lat".COut.Spin_Lat1.Work THEN #MB3_Decoder.OpDone := TRUE; END_IF;
END_REGION

REGION Network 22: MB3 Code 3044 - P5 - Sollevatori
   RUNG wire#powerrail
      { S7_Templates := "SrcType := Int" } EQ_Contact(in1 := #MB3_Decoder.Code, in2 := #"3044_SOLLEVATORI_P5")
      wire#w1
      Contact( #MB3_Decoder.OperationMinus )
      Coil( "A03_HMI".MB3.Button.A0301.SpintoreLat.Sollevatori.Rest )
   END_RUNG
   RUNG wire#w1
      Contact( #MB3_Decoder.OperationPlus )
      Coil( "A03_HMI".MB3.Button.A0301.SpintoreLat.Sollevatori.Work )
   END_RUNG
   RUNG wire#w1
      Contact( "A0301_Spintore_Lat".COut.Sollevatori.Rest_CheckNext )
      wire#w2
      S_Coil( #MB3_Decoder.OpEnabled )
   END_RUNG
   RUNG wire#w1
      Contact( "A0301_Spintore_Lat".COut.Sollevatori.Work_CheckNext )
   END_RUNG wire#w2
   RUNG wire#w1
      Contact( "A0301_Spintore_Lat".COut.Sollevatori.Rest )
      wire#w3
      I_Contact( "A0301_Spintore_Lat".COut.Sollevatori.Standstill )
      S_Coil( #MB3_Decoder.OpRunning )
   END_RUNG
   RUNG wire#w1
      Contact( "A0301_Spintore_Lat".COut.Sollevatori.Work )
   END_RUNG wire#w3
   RUNG wire#w1
      Contact( "A03_HMI".MB3.Button.A0301.SpintoreLat.Sollevatori.Rest )
      Contact( "A0301_Spintore_Lat".COut.Sollevatori.Rest )
      wire#w4
      Contact( "A0301_Spintore_Lat".COut.Sollevatori.Standstill )
      S_Coil( #MB3_Decoder.OpDone )
   END_RUNG
   RUNG wire#w1
      Contact( "A03_HMI".MB3.Button.A0301.SpintoreLat.Sollevatori.Work )
      Contact( "A0301_Spintore_Lat".COut.Sollevatori.Work )
   END_RUNG wire#w4
   // the same network as SCL:
   #_w1 := #MB3_Decoder.Code = #"3044_SOLLEVATORI_P5";
   "A03_HMI".MB3.Button.A0301.SpintoreLat.Sollevatori.Rest := #_w1 AND #MB3_Decoder.OperationMinus;
   "A03_HMI".MB3.Button.A0301.SpintoreLat.Sollevatori.Work := #_w1 AND #MB3_Decoder.OperationPlus;
   IF #_w1 AND ("A0301_Spintore_Lat".COut.Sollevatori.Rest_CheckNext OR "A0301_Spintore_Lat".COut.Sollevatori.Work_CheckNext) THEN
       #MB3_Decoder.OpEnabled := TRUE;
   END_IF;
   IF #_w1 AND ("A0301_Spintore_Lat".COut.Sollevatori.Rest OR "A0301_Spintore_Lat".COut.Sollevatori.Work) AND NOT "A0301_Spintore_Lat".COut.Sollevatori.Standstill THEN
       #MB3_Decoder.OpRunning := TRUE;
   END_IF;
   IF #_w1 AND (("A03_HMI".MB3.Button.A0301.SpintoreLat.Sollevatori.Rest AND "A0301_Spintore_Lat".COut.Sollevatori.Rest) OR ("A03_HMI".MB3.Button.A0301.SpintoreLat.Sollevatori.Work AND "A0301_Spintore_Lat".COut.Sollevatori.Work)) AND "A0301_Spintore_Lat".COut.Sollevatori.Standstill THEN
       #MB3_Decoder.OpDone := TRUE;
   END_IF;
END_REGION

REGION Network 23: <<<<<<<<< A0302 STAZIONE 2 >>>>>>>>>>>>>
END_REGION

REGION Network 24: MB3 Code 4001 - Area 03 HU Cytropack
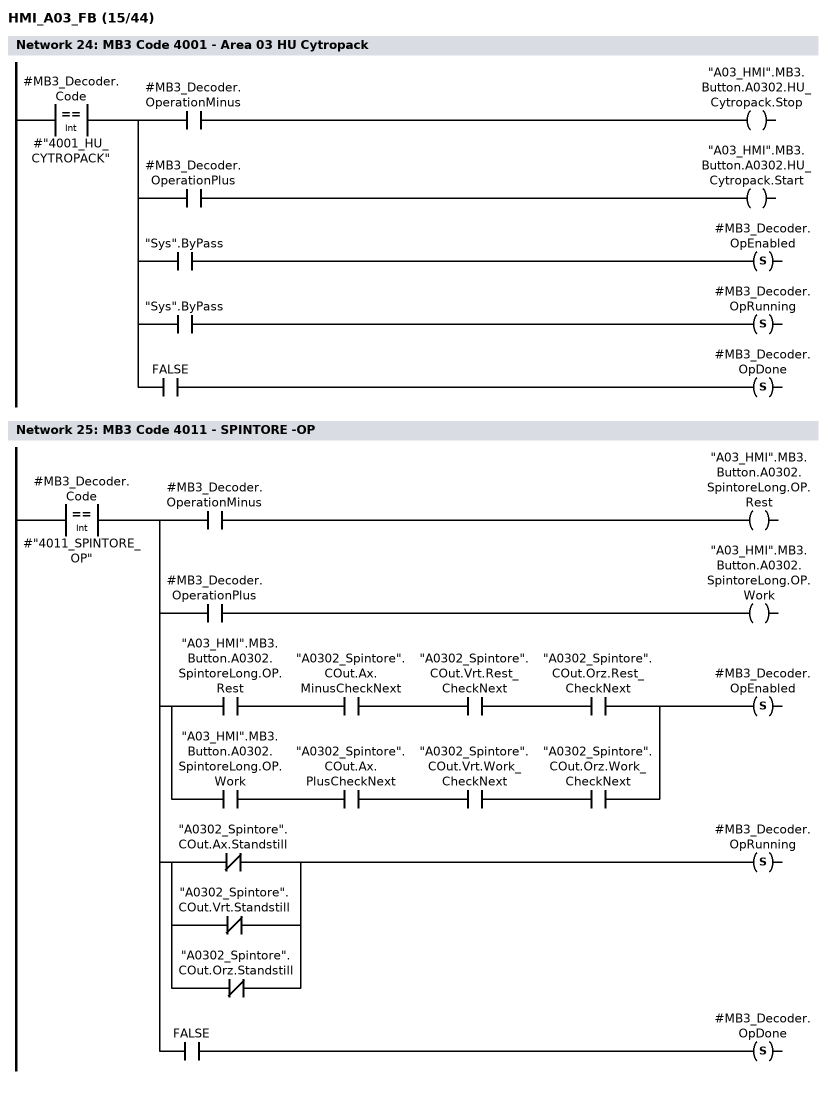
   RUNG wire#powerrail
      { S7_Templates := "SrcType := Int" } EQ_Contact(in1 := #MB3_Decoder.Code, in2 := #"4001_HU_CYTROPACK")
      wire#w1
      Contact( #MB3_Decoder.OperationMinus )
      Coil( "A03_HMI".MB3.Button.A0302.HU_Cytropack.Stop )
   END_RUNG
   RUNG wire#w1
      Contact( #MB3_Decoder.OperationPlus )
      Coil( "A03_HMI".MB3.Button.A0302.HU_Cytropack.Start )
   END_RUNG
   RUNG wire#w1
      Contact( "Sys".ByPass )
      S_Coil( #MB3_Decoder.OpEnabled )
   END_RUNG
   RUNG wire#w1
      Contact( "Sys".ByPass )
      S_Coil( #MB3_Decoder.OpRunning )
   END_RUNG
   RUNG wire#w1
      Contact( FALSE )
      S_Coil( #MB3_Decoder.OpDone )
   END_RUNG
   // the same network as SCL:
   #_w1 := #MB3_Decoder.Code = #"4001_HU_CYTROPACK";
   "A03_HMI".MB3.Button.A0302.HU_Cytropack.Stop := #_w1 AND #MB3_Decoder.OperationMinus;
   "A03_HMI".MB3.Button.A0302.HU_Cytropack.Start := #_w1 AND #MB3_Decoder.OperationPlus;
   IF #_w1 AND "Sys".ByPass THEN
       #MB3_Decoder.OpEnabled := TRUE;
       #MB3_Decoder.OpRunning := TRUE;
   END_IF;
   IF #_w1 AND FALSE THEN #MB3_Decoder.OpDone := TRUE; END_IF;
END_REGION

REGION Network 25: MB3 Code 4011 - SPINTORE -OP
   RUNG wire#powerrail
      { S7_Templates := "SrcType := Int" } EQ_Contact(in1 := #MB3_Decoder.Code, in2 := #"4011_SPINTORE_OP")
      wire#w1
      Contact( #MB3_Decoder.OperationMinus )
      Coil( "A03_HMI".MB3.Button.A0302.SpintoreLong.OP.Rest )
   END_RUNG
   RUNG wire#w1
      Contact( #MB3_Decoder.OperationPlus )
      Coil( "A03_HMI".MB3.Button.A0302.SpintoreLong.OP.Work )
   END_RUNG
   RUNG wire#w1
      Contact( "A03_HMI".MB3.Button.A0302.SpintoreLong.OP.Rest )
      Contact( "A0302_Spintore".COut.Ax.MinusCheckNext )
      Contact( "A0302_Spintore".COut.Vrt.Rest_CheckNext )
      Contact( "A0302_Spintore".COut.Orz.Rest_CheckNext )
      wire#w2
      S_Coil( #MB3_Decoder.OpEnabled )
   END_RUNG
   RUNG wire#w1
      Contact( "A03_HMI".MB3.Button.A0302.SpintoreLong.OP.Work )
      Contact( "A0302_Spintore".COut.Ax.PlusCheckNext )
      Contact( "A0302_Spintore".COut.Vrt.Work_CheckNext )
      Contact( "A0302_Spintore".COut.Orz.Work_CheckNext )
   END_RUNG wire#w2
   RUNG wire#w1
      I_Contact( "A0302_Spintore".COut.Ax.Standstill )
      wire#w3
      S_Coil( #MB3_Decoder.OpRunning )
   END_RUNG
   RUNG wire#w1
      I_Contact( "A0302_Spintore".COut.Vrt.Standstill )
   END_RUNG wire#w3
   RUNG wire#w1
      I_Contact( "A0302_Spintore".COut.Orz.Standstill )
   END_RUNG wire#w3
   RUNG wire#w1
      Contact( FALSE )
      S_Coil( #MB3_Decoder.OpDone )
   END_RUNG
   // the same network as SCL:
   #_w1 := #MB3_Decoder.Code = #"4011_SPINTORE_OP";
   "A03_HMI".MB3.Button.A0302.SpintoreLong.OP.Rest := #_w1 AND #MB3_Decoder.OperationMinus;
   "A03_HMI".MB3.Button.A0302.SpintoreLong.OP.Work := #_w1 AND #MB3_Decoder.OperationPlus;
   IF #_w1 AND (("A03_HMI".MB3.Button.A0302.SpintoreLong.OP.Rest AND "A0302_Spintore".COut.Ax.MinusCheckNext AND "A0302_Spintore".COut.Vrt.Rest_CheckNext AND "A0302_Spintore".COut.Orz.Rest_CheckNext) OR ("A03_HMI".MB3.Button.A0302.SpintoreLong.OP.Work AND "A0302_Spintore".COut.Ax.PlusCheckNext AND "A0302_Spintore".COut.Vrt.Work_CheckNext AND "A0302_Spintore".COut.Orz.Work_CheckNext)) THEN
       #MB3_Decoder.OpEnabled := TRUE;
   END_IF;
   IF #_w1 AND (NOT "A0302_Spintore".COut.Ax.Standstill OR NOT "A0302_Spintore".COut.Vrt.Standstill OR NOT "A0302_Spintore".COut.Orz.Standstill) THEN
       #MB3_Decoder.OpRunning := TRUE;
   END_IF;
   IF #_w1 AND FALSE THEN #MB3_Decoder.OpDone := TRUE; END_IF;
END_REGION

REGION Network 26: MB3 Code 4012 - SPINTORE -AX
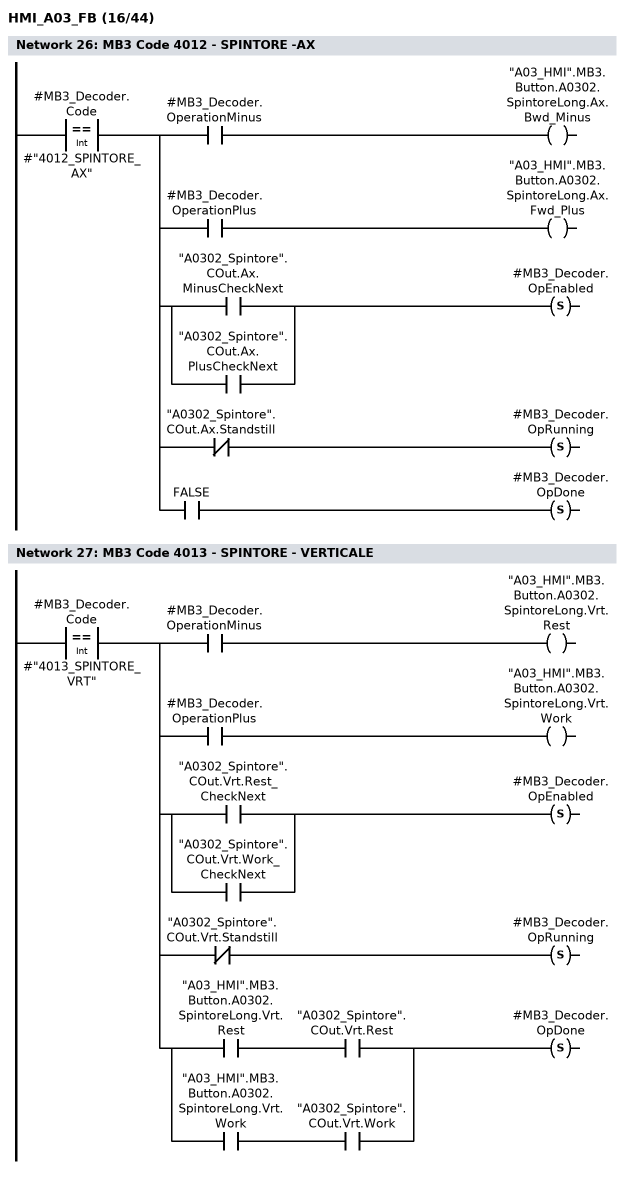
   RUNG wire#powerrail
      { S7_Templates := "SrcType := Int" } EQ_Contact(in1 := #MB3_Decoder.Code, in2 := #"4012_SPINTORE_AX")
      wire#w1
      Contact( #MB3_Decoder.OperationMinus )
      Coil( "A03_HMI".MB3.Button.A0302.SpintoreLong.Ax.Bwd_Minus )
   END_RUNG
   RUNG wire#w1
      Contact( #MB3_Decoder.OperationPlus )
      Coil( "A03_HMI".MB3.Button.A0302.SpintoreLong.Ax.Fwd_Plus )
   END_RUNG
   RUNG wire#w1
      Contact( "A0302_Spintore".COut.Ax.MinusCheckNext )
      wire#w2
      S_Coil( #MB3_Decoder.OpEnabled )
   END_RUNG
   RUNG wire#w1
      Contact( "A0302_Spintore".COut.Ax.PlusCheckNext )
   END_RUNG wire#w2
   RUNG wire#w1
      I_Contact( "A0302_Spintore".COut.Ax.Standstill )
      S_Coil( #MB3_Decoder.OpRunning )
   END_RUNG
   RUNG wire#w1
      Contact( FALSE )
      S_Coil( #MB3_Decoder.OpDone )
   END_RUNG
   // the same network as SCL:
   #_w1 := #MB3_Decoder.Code = #"4012_SPINTORE_AX";
   "A03_HMI".MB3.Button.A0302.SpintoreLong.Ax.Bwd_Minus := #_w1 AND #MB3_Decoder.OperationMinus;
   "A03_HMI".MB3.Button.A0302.SpintoreLong.Ax.Fwd_Plus := #_w1 AND #MB3_Decoder.OperationPlus;
   IF #_w1 AND ("A0302_Spintore".COut.Ax.MinusCheckNext OR "A0302_Spintore".COut.Ax.PlusCheckNext) THEN
       #MB3_Decoder.OpEnabled := TRUE;
   END_IF;
   IF #_w1 AND NOT "A0302_Spintore".COut.Ax.Standstill THEN #MB3_Decoder.OpRunning := TRUE; END_IF;
   IF #_w1 AND FALSE THEN #MB3_Decoder.OpDone := TRUE; END_IF;
END_REGION

REGION Network 27: MB3 Code 4013 - SPINTORE - VERTICALE
   RUNG wire#powerrail
      { S7_Templates := "SrcType := Int" } EQ_Contact(in1 := #MB3_Decoder.Code, in2 := #"4013_SPINTORE_VRT")
      wire#w1
      Contact( #MB3_Decoder.OperationMinus )
      Coil( "A03_HMI".MB3.Button.A0302.SpintoreLong.Vrt.Rest )
   END_RUNG
   RUNG wire#w1
      Contact( #MB3_Decoder.OperationPlus )
      Coil( "A03_HMI".MB3.Button.A0302.SpintoreLong.Vrt.Work )
   END_RUNG
   RUNG wire#w1
      Contact( "A0302_Spintore".COut.Vrt.Rest_CheckNext )
      wire#w2
      S_Coil( #MB3_Decoder.OpEnabled )
   END_RUNG
   RUNG wire#w1
      Contact( "A0302_Spintore".COut.Vrt.Work_CheckNext )
   END_RUNG wire#w2
   RUNG wire#w1
      I_Contact( "A0302_Spintore".COut.Vrt.Standstill )
      S_Coil( #MB3_Decoder.OpRunning )
   END_RUNG
   RUNG wire#w1
      Contact( "A03_HMI".MB3.Button.A0302.SpintoreLong.Vrt.Rest )
      Contact( "A0302_Spintore".COut.Vrt.Rest )
      wire#w3
      S_Coil( #MB3_Decoder.OpDone )
   END_RUNG
   RUNG wire#w1
      Contact( "A03_HMI".MB3.Button.A0302.SpintoreLong.Vrt.Work )
      Contact( "A0302_Spintore".COut.Vrt.Work )
   END_RUNG wire#w3
   // the same network as SCL:
   #_w1 := #MB3_Decoder.Code = #"4013_SPINTORE_VRT";
   "A03_HMI".MB3.Button.A0302.SpintoreLong.Vrt.Rest := #_w1 AND #MB3_Decoder.OperationMinus;
   "A03_HMI".MB3.Button.A0302.SpintoreLong.Vrt.Work := #_w1 AND #MB3_Decoder.OperationPlus;
   IF #_w1 AND ("A0302_Spintore".COut.Vrt.Rest_CheckNext OR "A0302_Spintore".COut.Vrt.Work_CheckNext) THEN
       #MB3_Decoder.OpEnabled := TRUE;
   END_IF;
   IF #_w1 AND NOT "A0302_Spintore".COut.Vrt.Standstill THEN #MB3_Decoder.OpRunning := TRUE; END_IF;
   IF #_w1 AND (("A03_HMI".MB3.Button.A0302.SpintoreLong.Vrt.Rest AND "A0302_Spintore".COut.Vrt.Rest) OR ("A03_HMI".MB3.Button.A0302.SpintoreLong.Vrt.Work AND "A0302_Spintore".COut.Vrt.Work)) THEN
       #MB3_Decoder.OpDone := TRUE;
   END_IF;
END_REGION

REGION Network 28: MB3 Code 4014 - SPINTORE - ORIZZONTALE
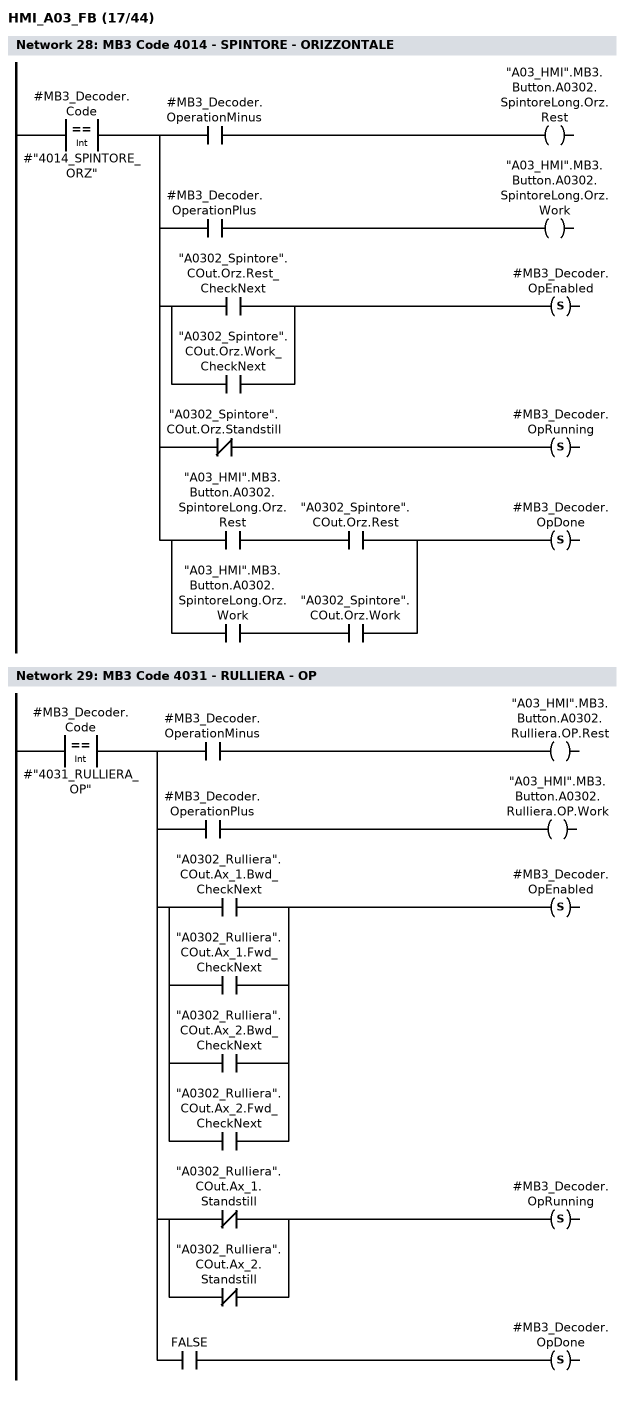
   RUNG wire#powerrail
      { S7_Templates := "SrcType := Int" } EQ_Contact(in1 := #MB3_Decoder.Code, in2 := #"4014_SPINTORE_ORZ")
      wire#w1
      Contact( #MB3_Decoder.OperationMinus )
      Coil( "A03_HMI".MB3.Button.A0302.SpintoreLong.Orz.Rest )
   END_RUNG
   RUNG wire#w1
      Contact( #MB3_Decoder.OperationPlus )
      Coil( "A03_HMI".MB3.Button.A0302.SpintoreLong.Orz.Work )
   END_RUNG
   RUNG wire#w1
      Contact( "A0302_Spintore".COut.Orz.Rest_CheckNext )
      wire#w2
      S_Coil( #MB3_Decoder.OpEnabled )
   END_RUNG
   RUNG wire#w1
      Contact( "A0302_Spintore".COut.Orz.Work_CheckNext )
   END_RUNG wire#w2
   RUNG wire#w1
      I_Contact( "A0302_Spintore".COut.Orz.Standstill )
      S_Coil( #MB3_Decoder.OpRunning )
   END_RUNG
   RUNG wire#w1
      Contact( "A03_HMI".MB3.Button.A0302.SpintoreLong.Orz.Rest )
      Contact( "A0302_Spintore".COut.Orz.Rest )
      wire#w3
      S_Coil( #MB3_Decoder.OpDone )
   END_RUNG
   RUNG wire#w1
      Contact( "A03_HMI".MB3.Button.A0302.SpintoreLong.Orz.Work )
      Contact( "A0302_Spintore".COut.Orz.Work )
   END_RUNG wire#w3
   // the same network as SCL:
   #_w1 := #MB3_Decoder.Code = #"4014_SPINTORE_ORZ";
   "A03_HMI".MB3.Button.A0302.SpintoreLong.Orz.Rest := #_w1 AND #MB3_Decoder.OperationMinus;
   "A03_HMI".MB3.Button.A0302.SpintoreLong.Orz.Work := #_w1 AND #MB3_Decoder.OperationPlus;
   IF #_w1 AND ("A0302_Spintore".COut.Orz.Rest_CheckNext OR "A0302_Spintore".COut.Orz.Work_CheckNext) THEN
       #MB3_Decoder.OpEnabled := TRUE;
   END_IF;
   IF #_w1 AND NOT "A0302_Spintore".COut.Orz.Standstill THEN #MB3_Decoder.OpRunning := TRUE; END_IF;
   IF #_w1 AND (("A03_HMI".MB3.Button.A0302.SpintoreLong.Orz.Rest AND "A0302_Spintore".COut.Orz.Rest) OR ("A03_HMI".MB3.Button.A0302.SpintoreLong.Orz.Work AND "A0302_Spintore".COut.Orz.Work)) THEN
       #MB3_Decoder.OpDone := TRUE;
   END_IF;
END_REGION

REGION Network 29: MB3 Code 4031 - RULLIERA - OP
   RUNG wire#powerrail
      { S7_Templates := "SrcType := Int" } EQ_Contact(in1 := #MB3_Decoder.Code, in2 := #"4031_RULLIERA_OP")
      wire#w1
      Contact( #MB3_Decoder.OperationMinus )
      Coil( "A03_HMI".MB3.Button.A0302.Rulliera.OP.Rest )
   END_RUNG
   RUNG wire#w1
      Contact( #MB3_Decoder.OperationPlus )
      Coil( "A03_HMI".MB3.Button.A0302.Rulliera.OP.Work )
   END_RUNG
   RUNG wire#w1
      Contact( "A0302_Rulliera".COut.Ax_1.Bwd_CheckNext )
      wire#w2
      S_Coil( #MB3_Decoder.OpEnabled )
   END_RUNG
   RUNG wire#w1
      Contact( "A0302_Rulliera".COut.Ax_1.Fwd_CheckNext )
   END_RUNG wire#w2
   RUNG wire#w1
      Contact( "A0302_Rulliera".COut.Ax_2.Bwd_CheckNext )
   END_RUNG wire#w2
   RUNG wire#w1
      Contact( "A0302_Rulliera".COut.Ax_2.Fwd_CheckNext )
   END_RUNG wire#w2
   RUNG wire#w1
      I_Contact( "A0302_Rulliera".COut.Ax_1.Standstill )
      wire#w3
      S_Coil( #MB3_Decoder.OpRunning )
   END_RUNG
   RUNG wire#w1
      I_Contact( "A0302_Rulliera".COut.Ax_2.Standstill )
   END_RUNG wire#w3
   RUNG wire#w1
      Contact( FALSE )
      S_Coil( #MB3_Decoder.OpDone )
   END_RUNG
   // the same network as SCL:
   #_w1 := #MB3_Decoder.Code = #"4031_RULLIERA_OP";
   "A03_HMI".MB3.Button.A0302.Rulliera.OP.Rest := #_w1 AND #MB3_Decoder.OperationMinus;
   "A03_HMI".MB3.Button.A0302.Rulliera.OP.Work := #_w1 AND #MB3_Decoder.OperationPlus;
   IF #_w1 AND ("A0302_Rulliera".COut.Ax_1.Bwd_CheckNext OR "A0302_Rulliera".COut.Ax_1.Fwd_CheckNext OR "A0302_Rulliera".COut.Ax_2.Bwd_CheckNext OR "A0302_Rulliera".COut.Ax_2.Fwd_CheckNext) THEN
       #MB3_Decoder.OpEnabled := TRUE;
   END_IF;
   IF #_w1 AND (NOT "A0302_Rulliera".COut.Ax_1.Standstill OR NOT "A0302_Rulliera".COut.Ax_2.Standstill) THEN
       #MB3_Decoder.OpRunning := TRUE;
   END_IF;
   IF #_w1 AND FALSE THEN #MB3_Decoder.OpDone := TRUE; END_IF;
END_REGION

REGION Network 30: MB3 Code 4032 - RULLIERA -AX
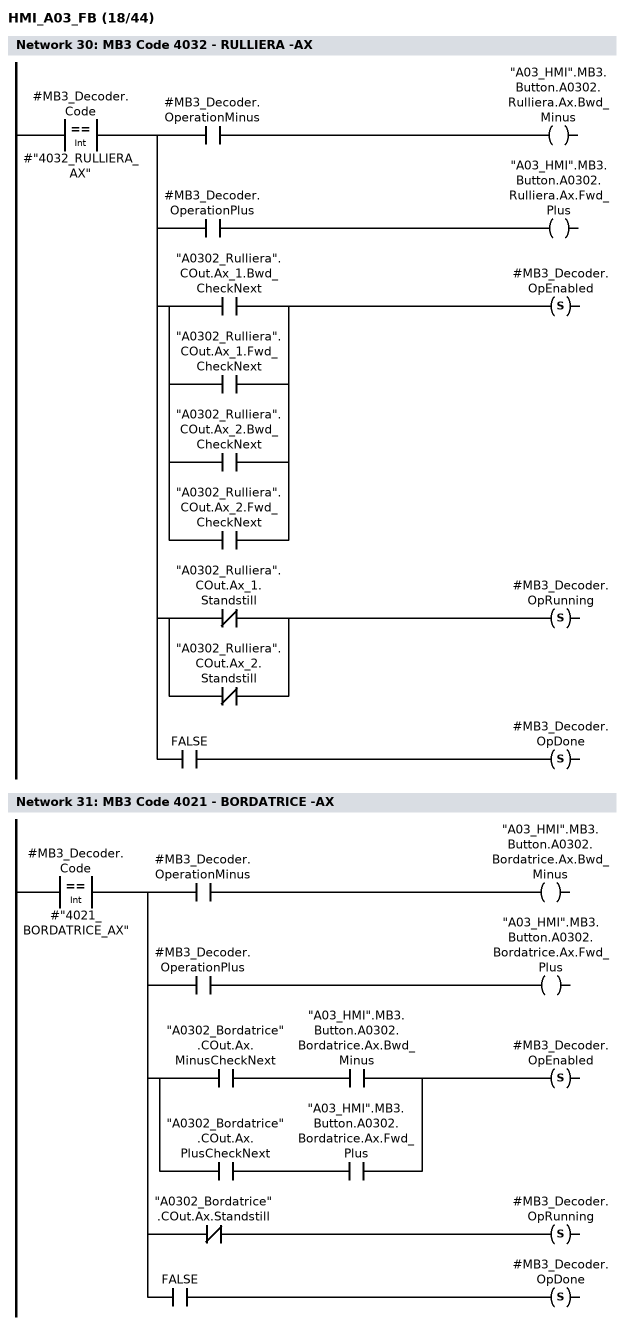
   RUNG wire#powerrail
      { S7_Templates := "SrcType := Int" } EQ_Contact(in1 := #MB3_Decoder.Code, in2 := #"4032_RULLIERA_AX")
      wire#w1
      Contact( #MB3_Decoder.OperationMinus )
      Coil( "A03_HMI".MB3.Button.A0302.Rulliera.Ax.Bwd_Minus )
   END_RUNG
   RUNG wire#w1
      Contact( #MB3_Decoder.OperationPlus )
      Coil( "A03_HMI".MB3.Button.A0302.Rulliera.Ax.Fwd_Plus )
   END_RUNG
   RUNG wire#w1
      Contact( "A0302_Rulliera".COut.Ax_1.Bwd_CheckNext )
      wire#w2
      S_Coil( #MB3_Decoder.OpEnabled )
   END_RUNG
   RUNG wire#w1
      Contact( "A0302_Rulliera".COut.Ax_1.Fwd_CheckNext )
   END_RUNG wire#w2
   RUNG wire#w1
      Contact( "A0302_Rulliera".COut.Ax_2.Bwd_CheckNext )
   END_RUNG wire#w2
   RUNG wire#w1
      Contact( "A0302_Rulliera".COut.Ax_2.Fwd_CheckNext )
   END_RUNG wire#w2
   RUNG wire#w1
      I_Contact( "A0302_Rulliera".COut.Ax_1.Standstill )
      wire#w3
      S_Coil( #MB3_Decoder.OpRunning )
   END_RUNG
   RUNG wire#w1
      I_Contact( "A0302_Rulliera".COut.Ax_2.Standstill )
   END_RUNG wire#w3
   RUNG wire#w1
      Contact( FALSE )
      S_Coil( #MB3_Decoder.OpDone )
   END_RUNG
   // the same network as SCL:
   #_w1 := #MB3_Decoder.Code = #"4032_RULLIERA_AX";
   "A03_HMI".MB3.Button.A0302.Rulliera.Ax.Bwd_Minus := #_w1 AND #MB3_Decoder.OperationMinus;
   "A03_HMI".MB3.Button.A0302.Rulliera.Ax.Fwd_Plus := #_w1 AND #MB3_Decoder.OperationPlus;
   IF #_w1 AND ("A0302_Rulliera".COut.Ax_1.Bwd_CheckNext OR "A0302_Rulliera".COut.Ax_1.Fwd_CheckNext OR "A0302_Rulliera".COut.Ax_2.Bwd_CheckNext OR "A0302_Rulliera".COut.Ax_2.Fwd_CheckNext) THEN
       #MB3_Decoder.OpEnabled := TRUE;
   END_IF;
   IF #_w1 AND (NOT "A0302_Rulliera".COut.Ax_1.Standstill OR NOT "A0302_Rulliera".COut.Ax_2.Standstill) THEN
       #MB3_Decoder.OpRunning := TRUE;
   END_IF;
   IF #_w1 AND FALSE THEN #MB3_Decoder.OpDone := TRUE; END_IF;
END_REGION

REGION Network 31: MB3 Code 4021 - BORDATRICE -AX
   RUNG wire#powerrail
      { S7_Templates := "SrcType := Int" } EQ_Contact(in1 := #MB3_Decoder.Code, in2 := #"4021_BORDATRICE_AX")
      wire#w1
      Contact( #MB3_Decoder.OperationMinus )
      Coil( "A03_HMI".MB3.Button.A0302.Bordatrice.Ax.Bwd_Minus )
   END_RUNG
   RUNG wire#w1
      Contact( #MB3_Decoder.OperationPlus )
      Coil( "A03_HMI".MB3.Button.A0302.Bordatrice.Ax.Fwd_Plus )
   END_RUNG
   RUNG wire#w1
      Contact( "A0302_Bordatrice".COut.Ax.MinusCheckNext )
      Contact( "A03_HMI".MB3.Button.A0302.Bordatrice.Ax.Bwd_Minus )
      wire#w2
      S_Coil( #MB3_Decoder.OpEnabled )
   END_RUNG
   RUNG wire#w1
      Contact( "A0302_Bordatrice".COut.Ax.PlusCheckNext )
      Contact( "A03_HMI".MB3.Button.A0302.Bordatrice.Ax.Fwd_Plus )
   END_RUNG wire#w2
   RUNG wire#w1
      I_Contact( "A0302_Bordatrice".COut.Ax.Standstill )
      S_Coil( #MB3_Decoder.OpRunning )
   END_RUNG
   RUNG wire#w1
      Contact( FALSE )
      S_Coil( #MB3_Decoder.OpDone )
   END_RUNG
   // the same network as SCL:
   #_w1 := #MB3_Decoder.Code = #"4021_BORDATRICE_AX";
   "A03_HMI".MB3.Button.A0302.Bordatrice.Ax.Bwd_Minus := #_w1 AND #MB3_Decoder.OperationMinus;
   "A03_HMI".MB3.Button.A0302.Bordatrice.Ax.Fwd_Plus := #_w1 AND #MB3_Decoder.OperationPlus;
   IF #_w1 AND (("A0302_Bordatrice".COut.Ax.MinusCheckNext AND "A03_HMI".MB3.Button.A0302.Bordatrice.Ax.Bwd_Minus) OR ("A0302_Bordatrice".COut.Ax.PlusCheckNext AND "A03_HMI".MB3.Button.A0302.Bordatrice.Ax.Fwd_Plus)) THEN
       #MB3_Decoder.OpEnabled := TRUE;
   END_IF;
   IF #_w1 AND NOT "A0302_Bordatrice".COut.Ax.Standstill THEN #MB3_Decoder.OpRunning := TRUE; END_IF;
   IF #_w1 AND FALSE THEN #MB3_Decoder.OpDone := TRUE; END_IF;
END_REGION

REGION Network 32: MB3 Code 4033 - REGOLAZ. BORDATRICE - CASSETTA
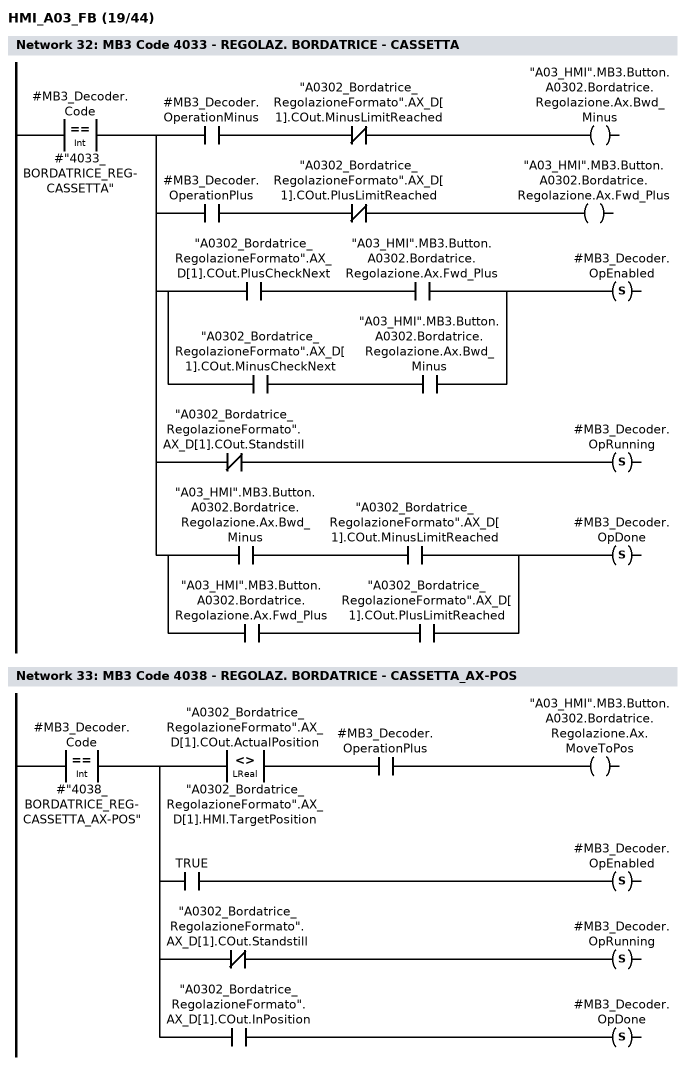
   RUNG wire#powerrail
      { S7_Templates := "SrcType := Int" } EQ_Contact(in1 := #MB3_Decoder.Code, in2 := #"4033_BORDATRICE_REG-CASSETTA")
      wire#w1
      Contact( #MB3_Decoder.OperationMinus )
      I_Contact( "A0302_Bordatrice_RegolazioneFormato".AX_D[1].COut.MinusLimitReached )
      Coil( "A03_HMI".MB3.Button.A0302.Bordatrice.Regolazione.Ax.Bwd_Minus )
   END_RUNG
   RUNG wire#w1
      Contact( #MB3_Decoder.OperationPlus )
      I_Contact( "A0302_Bordatrice_RegolazioneFormato".AX_D[1].COut.PlusLimitReached )
      Coil( "A03_HMI".MB3.Button.A0302.Bordatrice.Regolazione.Ax.Fwd_Plus )
   END_RUNG
   RUNG wire#w1
      Contact( "A0302_Bordatrice_RegolazioneFormato".AX_D[1].COut.PlusCheckNext )
      Contact( "A03_HMI".MB3.Button.A0302.Bordatrice.Regolazione.Ax.Fwd_Plus )
      wire#w2
      S_Coil( #MB3_Decoder.OpEnabled )
   END_RUNG
   RUNG wire#w1
      Contact( "A0302_Bordatrice_RegolazioneFormato".AX_D[1].COut.MinusCheckNext )
      Contact( "A03_HMI".MB3.Button.A0302.Bordatrice.Regolazione.Ax.Bwd_Minus )
   END_RUNG wire#w2
   RUNG wire#w1
      I_Contact( "A0302_Bordatrice_RegolazioneFormato".AX_D[1].COut.Standstill )
      S_Coil( #MB3_Decoder.OpRunning )
   END_RUNG
   RUNG wire#w1
      Contact( "A03_HMI".MB3.Button.A0302.Bordatrice.Regolazione.Ax.Bwd_Minus )
      Contact( "A0302_Bordatrice_RegolazioneFormato".AX_D[1].COut.MinusLimitReached )
      wire#w3
      S_Coil( #MB3_Decoder.OpDone )
   END_RUNG
   RUNG wire#w1
      Contact( "A03_HMI".MB3.Button.A0302.Bordatrice.Regolazione.Ax.Fwd_Plus )
      Contact( "A0302_Bordatrice_RegolazioneFormato".AX_D[1].COut.PlusLimitReached )
   END_RUNG wire#w3
   // the same network as SCL:
   #_w1 := #MB3_Decoder.Code = #"4033_BORDATRICE_REG-CASSETTA";
   "A03_HMI".MB3.Button.A0302.Bordatrice.Regolazione.Ax.Bwd_Minus := #_w1 AND #MB3_Decoder.OperationMinus AND NOT "A0302_Bordatrice_RegolazioneFormato".AX_D[1].COut.MinusLimitReached;
   "A03_HMI".MB3.Button.A0302.Bordatrice.Regolazione.Ax.Fwd_Plus := #_w1 AND #MB3_Decoder.OperationPlus AND NOT "A0302_Bordatrice_RegolazioneFormato".AX_D[1].COut.PlusLimitReached;
   IF #_w1 AND (("A0302_Bordatrice_RegolazioneFormato".AX_D[1].COut.PlusCheckNext AND "A03_HMI".MB3.Button.A0302.Bordatrice.Regolazione.Ax.Fwd_Plus) OR ("A0302_Bordatrice_RegolazioneFormato".AX_D[1].COut.MinusCheckNext AND "A03_HMI".MB3.Button.A0302.Bordatrice.Regolazione.Ax.Bwd_Minus)) THEN
       #MB3_Decoder.OpEnabled := TRUE;
   END_IF;
   IF #_w1 AND NOT "A0302_Bordatrice_RegolazioneFormato".AX_D[1].COut.Standstill THEN
       #MB3_Decoder.OpRunning := TRUE;
   END_IF;
   IF #_w1 AND (("A03_HMI".MB3.Button.A0302.Bordatrice.Regolazione.Ax.Bwd_Minus AND "A0302_Bordatrice_RegolazioneFormato".AX_D[1].COut.MinusLimitReached) OR ("A03_HMI".MB3.Button.A0302.Bordatrice.Regolazione.Ax.Fwd_Plus AND "A0302_Bordatrice_RegolazioneFormato".AX_D[1].COut.PlusLimitReached)) THEN
       #MB3_Decoder.OpDone := TRUE;
   END_IF;
END_REGION

REGION Network 33: MB3 Code 4038 - REGOLAZ. BORDATRICE - CASSETTA_AX-POS
   RUNG wire#powerrail
      { S7_Templates := "SrcType := Int" } EQ_Contact(in1 := #MB3_Decoder.Code, in2 := #"4038_BORDATRICE_REG-CASSETTA_AX-POS")
      wire#w1
      { S7_Templates := "SrcType := LReal" } NE_Contact(in1 := "A0302_Bordatrice_RegolazioneFormato".AX_D[1].COut.ActualPosition, in2 := "A0302_Bordatrice_RegolazioneFormato".AX_D[1].HMI.TargetPosition)
      Contact( #MB3_Decoder.OperationPlus )
      Coil( "A03_HMI".MB3.Button.A0302.Bordatrice.Regolazione.Ax.MoveToPos )
   END_RUNG
   RUNG wire#w1
      Contact( TRUE )
      S_Coil( #MB3_Decoder.OpEnabled )
   END_RUNG
   RUNG wire#w1
      I_Contact( "A0302_Bordatrice_RegolazioneFormato".AX_D[1].COut.Standstill )
      S_Coil( #MB3_Decoder.OpRunning )
   END_RUNG
   RUNG wire#w1
      Contact( "A0302_Bordatrice_RegolazioneFormato".AX_D[1].COut.InPosition )
      S_Coil( #MB3_Decoder.OpDone )
   END_RUNG
   // the same network as SCL:
   #_w1 := #MB3_Decoder.Code = #"4038_BORDATRICE_REG-CASSETTA_AX-POS";
   "A03_HMI".MB3.Button.A0302.Bordatrice.Regolazione.Ax.MoveToPos := #_w1 AND ("A0302_Bordatrice_RegolazioneFormato".AX_D[1].COut.ActualPosition <> "A0302_Bordatrice_RegolazioneFormato".AX_D[1].HMI.TargetPosition) AND #MB3_Decoder.OperationPlus;
   IF #_w1 AND TRUE THEN #MB3_Decoder.OpEnabled := TRUE; END_IF;
   IF #_w1 AND NOT "A0302_Bordatrice_RegolazioneFormato".AX_D[1].COut.Standstill THEN
       #MB3_Decoder.OpRunning := TRUE;
   END_IF;
   IF #_w1 AND "A0302_Bordatrice_RegolazioneFormato".AX_D[1].COut.InPosition THEN
       #MB3_Decoder.OpDone := TRUE;
   END_IF;
END_REGION

REGION Network 34: MB3 Code 4034 - REGOLAZ. BORDATRICE - PASSAGGIO 01 - COMBO
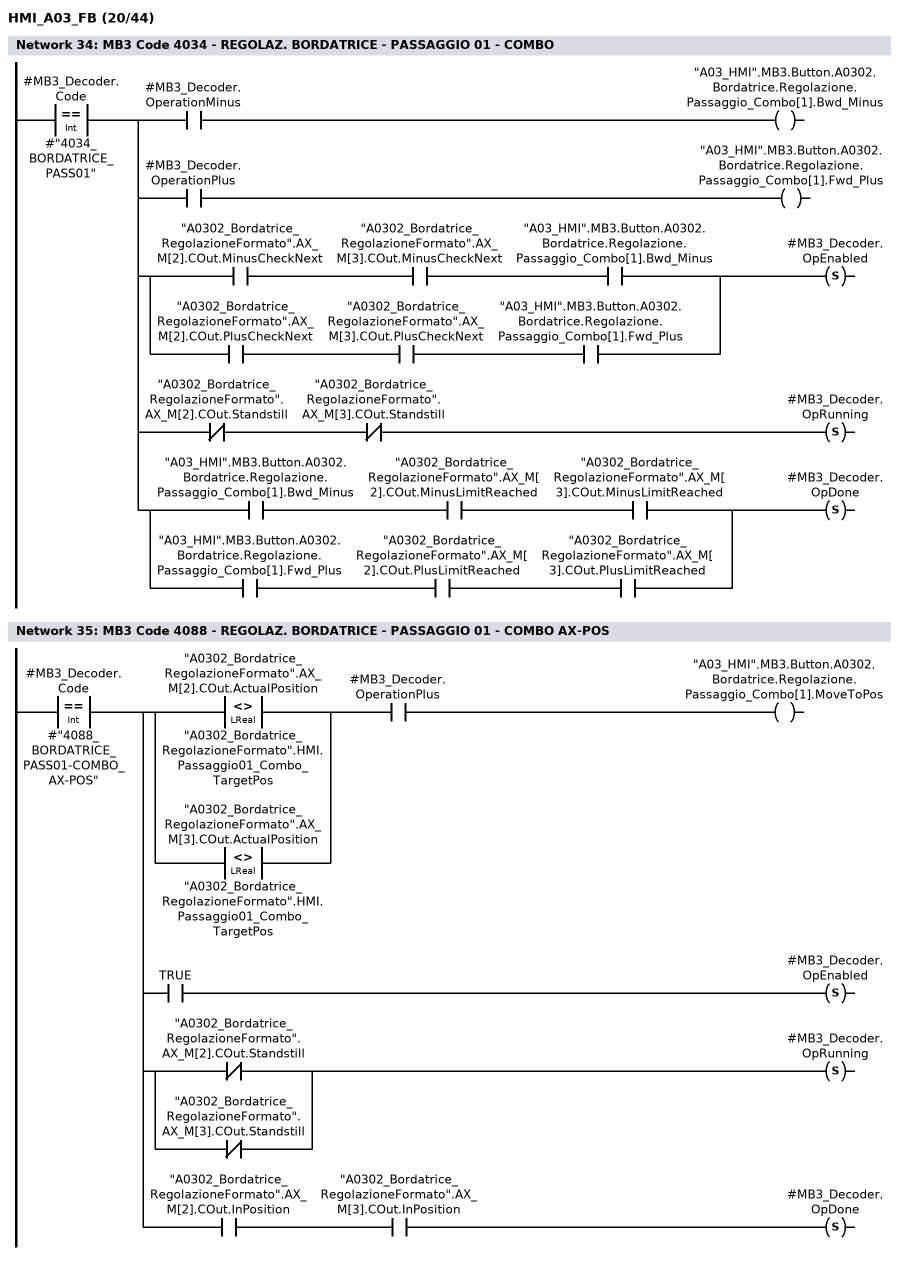
   RUNG wire#powerrail
      { S7_Templates := "SrcType := Int" } EQ_Contact(in1 := #MB3_Decoder.Code, in2 := #"4034_BORDATRICE_PASS01")
      wire#w1
      Contact( #MB3_Decoder.OperationMinus )
      Coil( "A03_HMI".MB3.Button.A0302.Bordatrice.Regolazione.Passaggio_Combo[1].Bwd_Minus )
   END_RUNG
   RUNG wire#w1
      Contact( #MB3_Decoder.OperationPlus )
      Coil( "A03_HMI".MB3.Button.A0302.Bordatrice.Regolazione.Passaggio_Combo[1].Fwd_Plus )
   END_RUNG
   RUNG wire#w1
      Contact( "A0302_Bordatrice_RegolazioneFormato".AX_M[2].COut.MinusCheckNext )
      Contact( "A0302_Bordatrice_RegolazioneFormato".AX_M[3].COut.MinusCheckNext )
      Contact( "A03_HMI".MB3.Button.A0302.Bordatrice.Regolazione.Passaggio_Combo[1].Bwd_Minus )
      wire#w2
      S_Coil( #MB3_Decoder.OpEnabled )
   END_RUNG
   RUNG wire#w1
      Contact( "A0302_Bordatrice_RegolazioneFormato".AX_M[2].COut.PlusCheckNext )
      Contact( "A0302_Bordatrice_RegolazioneFormato".AX_M[3].COut.PlusCheckNext )
      Contact( "A03_HMI".MB3.Button.A0302.Bordatrice.Regolazione.Passaggio_Combo[1].Fwd_Plus )
   END_RUNG wire#w2
   RUNG wire#w1
      I_Contact( "A0302_Bordatrice_RegolazioneFormato".AX_M[2].COut.Standstill )
      I_Contact( "A0302_Bordatrice_RegolazioneFormato".AX_M[3].COut.Standstill )
      S_Coil( #MB3_Decoder.OpRunning )
   END_RUNG
   RUNG wire#w1
      Contact( "A03_HMI".MB3.Button.A0302.Bordatrice.Regolazione.Passaggio_Combo[1].Bwd_Minus )
      Contact( "A0302_Bordatrice_RegolazioneFormato".AX_M[2].COut.MinusLimitReached )
      Contact( "A0302_Bordatrice_RegolazioneFormato".AX_M[3].COut.MinusLimitReached )
      wire#w3
      S_Coil( #MB3_Decoder.OpDone )
   END_RUNG
   RUNG wire#w1
      Contact( "A03_HMI".MB3.Button.A0302.Bordatrice.Regolazione.Passaggio_Combo[1].Fwd_Plus )
      Contact( "A0302_Bordatrice_RegolazioneFormato".AX_M[2].COut.PlusLimitReached )
      Contact( "A0302_Bordatrice_RegolazioneFormato".AX_M[3].COut.PlusLimitReached )
   END_RUNG wire#w3
   // the same network as SCL:
   #_w1 := #MB3_Decoder.Code = #"4034_BORDATRICE_PASS01";
   "A03_HMI".MB3.Button.A0302.Bordatrice.Regolazione.Passaggio_Combo[1].Bwd_Minus := #_w1 AND #MB3_Decoder.OperationMinus;
   "A03_HMI".MB3.Button.A0302.Bordatrice.Regolazione.Passaggio_Combo[1].Fwd_Plus := #_w1 AND #MB3_Decoder.OperationPlus;
   IF #_w1 AND (("A0302_Bordatrice_RegolazioneFormato".AX_M[2].COut.MinusCheckNext AND "A0302_Bordatrice_RegolazioneFormato".AX_M[3].COut.MinusCheckNext AND "A03_HMI".MB3.Button.A0302.Bordatrice.Regolazione.Passaggio_Combo[1].Bwd_Minus) OR ("A0302_Bordatrice_RegolazioneFormato".AX_M[2].COut.PlusCheckNext AND "A0302_Bordatrice_RegolazioneFormato".AX_M[3].COut.PlusCheckNext AND "A03_HMI".MB3.Button.A0302.Bordatrice.Regolazione.Passaggio_Combo[1].Fwd_Plus)) THEN
       #MB3_Decoder.OpEnabled := TRUE;
   END_IF;
   IF #_w1 AND NOT "A0302_Bordatrice_RegolazioneFormato".AX_M[2].COut.Standstill AND NOT "A0302_Bordatrice_RegolazioneFormato".AX_M[3].COut.Standstill THEN
       #MB3_Decoder.OpRunning := TRUE;
   END_IF;
   IF #_w1 AND (("A03_HMI".MB3.Button.A0302.Bordatrice.Regolazione.Passaggio_Combo[1].Bwd_Minus AND "A0302_Bordatrice_RegolazioneFormato".AX_M[2].COut.MinusLimitReached AND "A0302_Bordatrice_RegolazioneFormato".AX_M[3].COut.MinusLimitReached) OR ("A03_HMI".MB3.Button.A0302.Bordatrice.Regolazione.Passaggio_Combo[1].Fwd_Plus AND "A0302_Bordatrice_RegolazioneFormato".AX_M[2].COut.PlusLimitReached AND "A0302_Bordatrice_RegolazioneFormato".AX_M[3].COut.PlusLimitReached)) THEN
       #MB3_Decoder.OpDone := TRUE;
   END_IF;
END_REGION

REGION Network 35: MB3 Code 4088 - REGOLAZ. BORDATRICE - PASSAGGIO 01 - COMBO AX-POS
   RUNG wire#powerrail
      { S7_Templates := "SrcType := Int" } EQ_Contact(in1 := #MB3_Decoder.Code, in2 := #"4088_BORDATRICE_PASS01-COMBO_AX-POS")
      wire#w1
      { S7_Templates := "SrcType := LReal" } NE_Contact(in1 := "A0302_Bordatrice_RegolazioneFormato".AX_M[2].COut.ActualPosition, in2 := "A0302_Bordatrice_RegolazioneFormato".HMI.Passaggio01_Combo_TargetPos)
      wire#w2
      Contact( #MB3_Decoder.OperationPlus )
      Coil( "A03_HMI".MB3.Button.A0302.Bordatrice.Regolazione.Passaggio_Combo[1].MoveToPos )
   END_RUNG
   RUNG wire#w1
      { S7_Templates := "SrcType := LReal" } NE_Contact(in1 := "A0302_Bordatrice_RegolazioneFormato".AX_M[3].COut.ActualPosition, in2 := "A0302_Bordatrice_RegolazioneFormato".HMI.Passaggio01_Combo_TargetPos)
   END_RUNG wire#w2
   RUNG wire#w1
      Contact( TRUE )
      S_Coil( #MB3_Decoder.OpEnabled )
   END_RUNG
   RUNG wire#w1
      I_Contact( "A0302_Bordatrice_RegolazioneFormato".AX_M[2].COut.Standstill )
      wire#w3
      S_Coil( #MB3_Decoder.OpRunning )
   END_RUNG
   RUNG wire#w1
      I_Contact( "A0302_Bordatrice_RegolazioneFormato".AX_M[3].COut.Standstill )
   END_RUNG wire#w3
   RUNG wire#w1
      Contact( "A0302_Bordatrice_RegolazioneFormato".AX_M[2].COut.InPosition )
      Contact( "A0302_Bordatrice_RegolazioneFormato".AX_M[3].COut.InPosition )
      S_Coil( #MB3_Decoder.OpDone )
   END_RUNG
   // the same network as SCL:
   #_w1 := #MB3_Decoder.Code = #"4088_BORDATRICE_PASS01-COMBO_AX-POS";
   "A03_HMI".MB3.Button.A0302.Bordatrice.Regolazione.Passaggio_Combo[1].MoveToPos := #_w1 AND (("A0302_Bordatrice_RegolazioneFormato".AX_M[2].COut.ActualPosition <> "A0302_Bordatrice_RegolazioneFormato".HMI.Passaggio01_Combo_TargetPos) OR ("A0302_Bordatrice_RegolazioneFormato".AX_M[3].COut.ActualPosition <> "A0302_Bordatrice_RegolazioneFormato".HMI.Passaggio01_Combo_TargetPos)) AND #MB3_Decoder.OperationPlus;
   IF #_w1 AND TRUE THEN #MB3_Decoder.OpEnabled := TRUE; END_IF;
   IF #_w1 AND (NOT "A0302_Bordatrice_RegolazioneFormato".AX_M[2].COut.Standstill OR NOT "A0302_Bordatrice_RegolazioneFormato".AX_M[3].COut.Standstill) THEN
       #MB3_Decoder.OpRunning := TRUE;
   END_IF;
   IF #_w1 AND "A0302_Bordatrice_RegolazioneFormato".AX_M[2].COut.InPosition AND "A0302_Bordatrice_RegolazioneFormato".AX_M[3].COut.InPosition THEN
       #MB3_Decoder.OpDone := TRUE;
   END_IF;
END_REGION

REGION Network 36: MB3 Code 4080 - REGOLAZ. BORDATRICE - PASSAGGIO 01 - LATO-OP
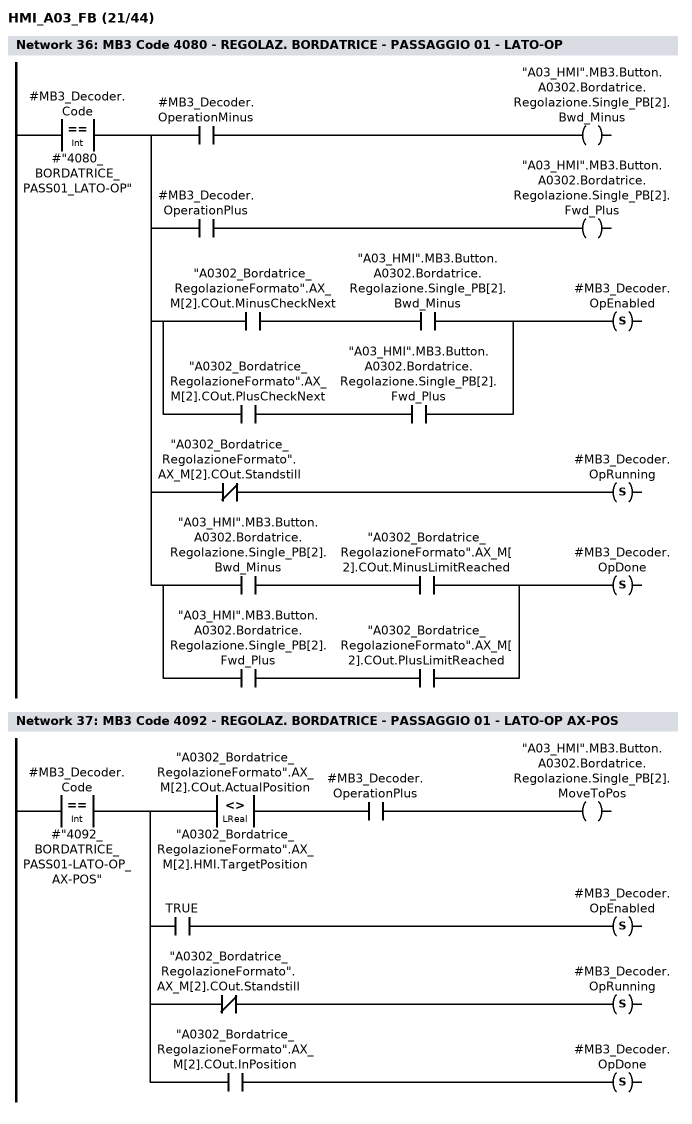
   RUNG wire#powerrail
      { S7_Templates := "SrcType := Int" } EQ_Contact(in1 := #MB3_Decoder.Code, in2 := #"4080_BORDATRICE_PASS01_LATO-OP")
      wire#w1
      Contact( #MB3_Decoder.OperationMinus )
      Coil( "A03_HMI".MB3.Button.A0302.Bordatrice.Regolazione.Single_PB[2].Bwd_Minus )
   END_RUNG
   RUNG wire#w1
      Contact( #MB3_Decoder.OperationPlus )
      Coil( "A03_HMI".MB3.Button.A0302.Bordatrice.Regolazione.Single_PB[2].Fwd_Plus )
   END_RUNG
   RUNG wire#w1
      Contact( "A0302_Bordatrice_RegolazioneFormato".AX_M[2].COut.MinusCheckNext )
      Contact( "A03_HMI".MB3.Button.A0302.Bordatrice.Regolazione.Single_PB[2].Bwd_Minus )
      wire#w2
      S_Coil( #MB3_Decoder.OpEnabled )
   END_RUNG
   RUNG wire#w1
      Contact( "A0302_Bordatrice_RegolazioneFormato".AX_M[2].COut.PlusCheckNext )
      Contact( "A03_HMI".MB3.Button.A0302.Bordatrice.Regolazione.Single_PB[2].Fwd_Plus )
   END_RUNG wire#w2
   RUNG wire#w1
      I_Contact( "A0302_Bordatrice_RegolazioneFormato".AX_M[2].COut.Standstill )
      S_Coil( #MB3_Decoder.OpRunning )
   END_RUNG
   RUNG wire#w1
      Contact( "A03_HMI".MB3.Button.A0302.Bordatrice.Regolazione.Single_PB[2].Bwd_Minus )
      Contact( "A0302_Bordatrice_RegolazioneFormato".AX_M[2].COut.MinusLimitReached )
      wire#w3
      S_Coil( #MB3_Decoder.OpDone )
   END_RUNG
   RUNG wire#w1
      Contact( "A03_HMI".MB3.Button.A0302.Bordatrice.Regolazione.Single_PB[2].Fwd_Plus )
      Contact( "A0302_Bordatrice_RegolazioneFormato".AX_M[2].COut.PlusLimitReached )
   END_RUNG wire#w3
   // the same network as SCL:
   #_w1 := #MB3_Decoder.Code = #"4080_BORDATRICE_PASS01_LATO-OP";
   "A03_HMI".MB3.Button.A0302.Bordatrice.Regolazione.Single_PB[2].Bwd_Minus := #_w1 AND #MB3_Decoder.OperationMinus;
   "A03_HMI".MB3.Button.A0302.Bordatrice.Regolazione.Single_PB[2].Fwd_Plus := #_w1 AND #MB3_Decoder.OperationPlus;
   IF #_w1 AND (("A0302_Bordatrice_RegolazioneFormato".AX_M[2].COut.MinusCheckNext AND "A03_HMI".MB3.Button.A0302.Bordatrice.Regolazione.Single_PB[2].Bwd_Minus) OR ("A0302_Bordatrice_RegolazioneFormato".AX_M[2].COut.PlusCheckNext AND "A03_HMI".MB3.Button.A0302.Bordatrice.Regolazione.Single_PB[2].Fwd_Plus)) THEN
       #MB3_Decoder.OpEnabled := TRUE;
   END_IF;
   IF #_w1 AND NOT "A0302_Bordatrice_RegolazioneFormato".AX_M[2].COut.Standstill THEN
       #MB3_Decoder.OpRunning := TRUE;
   END_IF;
   IF #_w1 AND (("A03_HMI".MB3.Button.A0302.Bordatrice.Regolazione.Single_PB[2].Bwd_Minus AND "A0302_Bordatrice_RegolazioneFormato".AX_M[2].COut.MinusLimitReached) OR ("A03_HMI".MB3.Button.A0302.Bordatrice.Regolazione.Single_PB[2].Fwd_Plus AND "A0302_Bordatrice_RegolazioneFormato".AX_M[2].COut.PlusLimitReached)) THEN
       #MB3_Decoder.OpDone := TRUE;
   END_IF;
END_REGION

REGION Network 37: MB3 Code 4092 - REGOLAZ. BORDATRICE - PASSAGGIO 01 - LATO-OP AX-POS
   RUNG wire#powerrail
      { S7_Templates := "SrcType := Int" } EQ_Contact(in1 := #MB3_Decoder.Code, in2 := #"4092_BORDATRICE_PASS01-LATO-OP_AX-POS")
      wire#w1
      { S7_Templates := "SrcType := LReal" } NE_Contact(in1 := "A0302_Bordatrice_RegolazioneFormato".AX_M[2].COut.ActualPosition, in2 := "A0302_Bordatrice_RegolazioneFormato".AX_M[2].HMI.TargetPosition)
      Contact( #MB3_Decoder.OperationPlus )
      Coil( "A03_HMI".MB3.Button.A0302.Bordatrice.Regolazione.Single_PB[2].MoveToPos )
   END_RUNG
   RUNG wire#w1
      Contact( TRUE )
      S_Coil( #MB3_Decoder.OpEnabled )
   END_RUNG
   RUNG wire#w1
      I_Contact( "A0302_Bordatrice_RegolazioneFormato".AX_M[2].COut.Standstill )
      S_Coil( #MB3_Decoder.OpRunning )
   END_RUNG
   RUNG wire#w1
      Contact( "A0302_Bordatrice_RegolazioneFormato".AX_M[2].COut.InPosition )
      S_Coil( #MB3_Decoder.OpDone )
   END_RUNG
   // the same network as SCL:
   #_w1 := #MB3_Decoder.Code = #"4092_BORDATRICE_PASS01-LATO-OP_AX-POS";
   "A03_HMI".MB3.Button.A0302.Bordatrice.Regolazione.Single_PB[2].MoveToPos := #_w1 AND ("A0302_Bordatrice_RegolazioneFormato".AX_M[2].COut.ActualPosition <> "A0302_Bordatrice_RegolazioneFormato".AX_M[2].HMI.TargetPosition) AND #MB3_Decoder.OperationPlus;
   IF #_w1 AND TRUE THEN #MB3_Decoder.OpEnabled := TRUE; END_IF;
   IF #_w1 AND NOT "A0302_Bordatrice_RegolazioneFormato".AX_M[2].COut.Standstill THEN
       #MB3_Decoder.OpRunning := TRUE;
   END_IF;
   IF #_w1 AND "A0302_Bordatrice_RegolazioneFormato".AX_M[2].COut.InPosition THEN
       #MB3_Decoder.OpDone := TRUE;
   END_IF;
END_REGION

REGION Network 38: MB3 Code 4081 - REGOLAZ. BORDATRICE - PASSAGGIO 01 - LATO-MOT
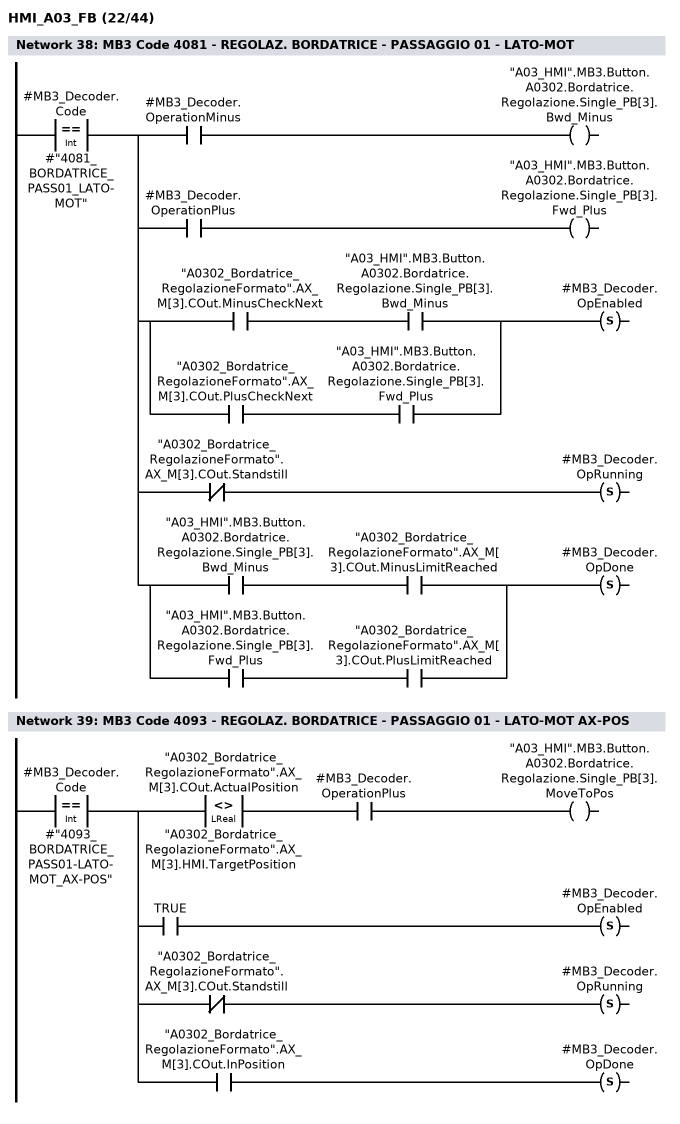
   RUNG wire#powerrail
      { S7_Templates := "SrcType := Int" } EQ_Contact(in1 := #MB3_Decoder.Code, in2 := #"4081_BORDATRICE_PASS01_LATO-MOT")
      wire#w1
      Contact( #MB3_Decoder.OperationMinus )
      Coil( "A03_HMI".MB3.Button.A0302.Bordatrice.Regolazione.Single_PB[3].Bwd_Minus )
   END_RUNG
   RUNG wire#w1
      Contact( #MB3_Decoder.OperationPlus )
      Coil( "A03_HMI".MB3.Button.A0302.Bordatrice.Regolazione.Single_PB[3].Fwd_Plus )
   END_RUNG
   RUNG wire#w1
      Contact( "A0302_Bordatrice_RegolazioneFormato".AX_M[3].COut.MinusCheckNext )
      Contact( "A03_HMI".MB3.Button.A0302.Bordatrice.Regolazione.Single_PB[3].Bwd_Minus )
      wire#w2
      S_Coil( #MB3_Decoder.OpEnabled )
   END_RUNG
   RUNG wire#w1
      Contact( "A0302_Bordatrice_RegolazioneFormato".AX_M[3].COut.PlusCheckNext )
      Contact( "A03_HMI".MB3.Button.A0302.Bordatrice.Regolazione.Single_PB[3].Fwd_Plus )
   END_RUNG wire#w2
   RUNG wire#w1
      I_Contact( "A0302_Bordatrice_RegolazioneFormato".AX_M[3].COut.Standstill )
      S_Coil( #MB3_Decoder.OpRunning )
   END_RUNG
   RUNG wire#w1
      Contact( "A03_HMI".MB3.Button.A0302.Bordatrice.Regolazione.Single_PB[3].Bwd_Minus )
      Contact( "A0302_Bordatrice_RegolazioneFormato".AX_M[3].COut.MinusLimitReached )
      wire#w3
      S_Coil( #MB3_Decoder.OpDone )
   END_RUNG
   RUNG wire#w1
      Contact( "A03_HMI".MB3.Button.A0302.Bordatrice.Regolazione.Single_PB[3].Fwd_Plus )
      Contact( "A0302_Bordatrice_RegolazioneFormato".AX_M[3].COut.PlusLimitReached )
   END_RUNG wire#w3
   // the same network as SCL:
   #_w1 := #MB3_Decoder.Code = #"4081_BORDATRICE_PASS01_LATO-MOT";
   "A03_HMI".MB3.Button.A0302.Bordatrice.Regolazione.Single_PB[3].Bwd_Minus := #_w1 AND #MB3_Decoder.OperationMinus;
   "A03_HMI".MB3.Button.A0302.Bordatrice.Regolazione.Single_PB[3].Fwd_Plus := #_w1 AND #MB3_Decoder.OperationPlus;
   IF #_w1 AND (("A0302_Bordatrice_RegolazioneFormato".AX_M[3].COut.MinusCheckNext AND "A03_HMI".MB3.Button.A0302.Bordatrice.Regolazione.Single_PB[3].Bwd_Minus) OR ("A0302_Bordatrice_RegolazioneFormato".AX_M[3].COut.PlusCheckNext AND "A03_HMI".MB3.Button.A0302.Bordatrice.Regolazione.Single_PB[3].Fwd_Plus)) THEN
       #MB3_Decoder.OpEnabled := TRUE;
   END_IF;
   IF #_w1 AND NOT "A0302_Bordatrice_RegolazioneFormato".AX_M[3].COut.Standstill THEN
       #MB3_Decoder.OpRunning := TRUE;
   END_IF;
   IF #_w1 AND (("A03_HMI".MB3.Button.A0302.Bordatrice.Regolazione.Single_PB[3].Bwd_Minus AND "A0302_Bordatrice_RegolazioneFormato".AX_M[3].COut.MinusLimitReached) OR ("A03_HMI".MB3.Button.A0302.Bordatrice.Regolazione.Single_PB[3].Fwd_Plus AND "A0302_Bordatrice_RegolazioneFormato".AX_M[3].COut.PlusLimitReached)) THEN
       #MB3_Decoder.OpDone := TRUE;
   END_IF;
END_REGION

REGION Network 39: MB3 Code 4093 - REGOLAZ. BORDATRICE - PASSAGGIO 01 - LATO-MOT AX-POS
   RUNG wire#powerrail
      { S7_Templates := "SrcType := Int" } EQ_Contact(in1 := #MB3_Decoder.Code, in2 := #"4093_BORDATRICE_PASS01-LATO-MOT_AX-POS")
      wire#w1
      { S7_Templates := "SrcType := LReal" } NE_Contact(in1 := "A0302_Bordatrice_RegolazioneFormato".AX_M[3].COut.ActualPosition, in2 := "A0302_Bordatrice_RegolazioneFormato".AX_M[3].HMI.TargetPosition)
      Contact( #MB3_Decoder.OperationPlus )
      Coil( "A03_HMI".MB3.Button.A0302.Bordatrice.Regolazione.Single_PB[3].MoveToPos )
   END_RUNG
   RUNG wire#w1
      Contact( TRUE )
      S_Coil( #MB3_Decoder.OpEnabled )
   END_RUNG
   RUNG wire#w1
      I_Contact( "A0302_Bordatrice_RegolazioneFormato".AX_M[3].COut.Standstill )
      S_Coil( #MB3_Decoder.OpRunning )
   END_RUNG
   RUNG wire#w1
      Contact( "A0302_Bordatrice_RegolazioneFormato".AX_M[3].COut.InPosition )
      S_Coil( #MB3_Decoder.OpDone )
   END_RUNG
   // the same network as SCL:
   #_w1 := #MB3_Decoder.Code = #"4093_BORDATRICE_PASS01-LATO-MOT_AX-POS";
   "A03_HMI".MB3.Button.A0302.Bordatrice.Regolazione.Single_PB[3].MoveToPos := #_w1 AND ("A0302_Bordatrice_RegolazioneFormato".AX_M[3].COut.ActualPosition <> "A0302_Bordatrice_RegolazioneFormato".AX_M[3].HMI.TargetPosition) AND #MB3_Decoder.OperationPlus;
   IF #_w1 AND TRUE THEN #MB3_Decoder.OpEnabled := TRUE; END_IF;
   IF #_w1 AND NOT "A0302_Bordatrice_RegolazioneFormato".AX_M[3].COut.Standstill THEN
       #MB3_Decoder.OpRunning := TRUE;
   END_IF;
   IF #_w1 AND "A0302_Bordatrice_RegolazioneFormato".AX_M[3].COut.InPosition THEN
       #MB3_Decoder.OpDone := TRUE;
   END_IF;
END_REGION

REGION Network 40: MB3 Code 4035 - REGOLAZ. BORDATRICE - PASSAGGIO 02 - COMBO
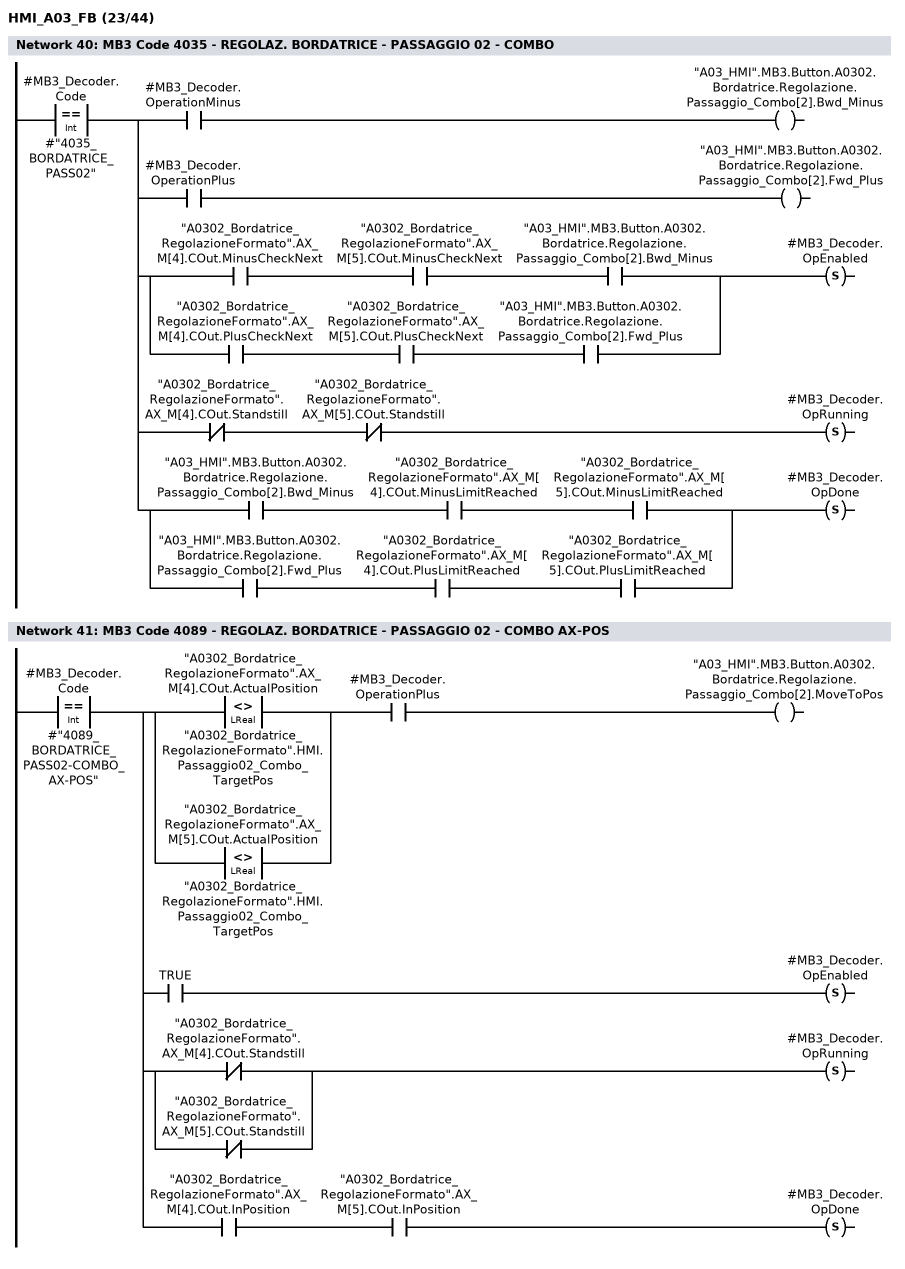
   RUNG wire#powerrail
      { S7_Templates := "SrcType := Int" } EQ_Contact(in1 := #MB3_Decoder.Code, in2 := #"4035_BORDATRICE_PASS02")
      wire#w1
      Contact( #MB3_Decoder.OperationMinus )
      Coil( "A03_HMI".MB3.Button.A0302.Bordatrice.Regolazione.Passaggio_Combo[2].Bwd_Minus )
   END_RUNG
   RUNG wire#w1
      Contact( #MB3_Decoder.OperationPlus )
      Coil( "A03_HMI".MB3.Button.A0302.Bordatrice.Regolazione.Passaggio_Combo[2].Fwd_Plus )
   END_RUNG
   RUNG wire#w1
      Contact( "A0302_Bordatrice_RegolazioneFormato".AX_M[4].COut.MinusCheckNext )
      Contact( "A0302_Bordatrice_RegolazioneFormato".AX_M[5].COut.MinusCheckNext )
      Contact( "A03_HMI".MB3.Button.A0302.Bordatrice.Regolazione.Passaggio_Combo[2].Bwd_Minus )
      wire#w2
      S_Coil( #MB3_Decoder.OpEnabled )
   END_RUNG
   RUNG wire#w1
      Contact( "A0302_Bordatrice_RegolazioneFormato".AX_M[4].COut.PlusCheckNext )
      Contact( "A0302_Bordatrice_RegolazioneFormato".AX_M[5].COut.PlusCheckNext )
      Contact( "A03_HMI".MB3.Button.A0302.Bordatrice.Regolazione.Passaggio_Combo[2].Fwd_Plus )
   END_RUNG wire#w2
   RUNG wire#w1
      I_Contact( "A0302_Bordatrice_RegolazioneFormato".AX_M[4].COut.Standstill )
      I_Contact( "A0302_Bordatrice_RegolazioneFormato".AX_M[5].COut.Standstill )
      S_Coil( #MB3_Decoder.OpRunning )
   END_RUNG
   RUNG wire#w1
      Contact( "A03_HMI".MB3.Button.A0302.Bordatrice.Regolazione.Passaggio_Combo[2].Bwd_Minus )
      Contact( "A0302_Bordatrice_RegolazioneFormato".AX_M[4].COut.MinusLimitReached )
      Contact( "A0302_Bordatrice_RegolazioneFormato".AX_M[5].COut.MinusLimitReached )
      wire#w3
      S_Coil( #MB3_Decoder.OpDone )
   END_RUNG
   RUNG wire#w1
      Contact( "A03_HMI".MB3.Button.A0302.Bordatrice.Regolazione.Passaggio_Combo[2].Fwd_Plus )
      Contact( "A0302_Bordatrice_RegolazioneFormato".AX_M[4].COut.PlusLimitReached )
      Contact( "A0302_Bordatrice_RegolazioneFormato".AX_M[5].COut.PlusLimitReached )
   END_RUNG wire#w3
   // the same network as SCL:
   #_w1 := #MB3_Decoder.Code = #"4035_BORDATRICE_PASS02";
   "A03_HMI".MB3.Button.A0302.Bordatrice.Regolazione.Passaggio_Combo[2].Bwd_Minus := #_w1 AND #MB3_Decoder.OperationMinus;
   "A03_HMI".MB3.Button.A0302.Bordatrice.Regolazione.Passaggio_Combo[2].Fwd_Plus := #_w1 AND #MB3_Decoder.OperationPlus;
   IF #_w1 AND (("A0302_Bordatrice_RegolazioneFormato".AX_M[4].COut.MinusCheckNext AND "A0302_Bordatrice_RegolazioneFormato".AX_M[5].COut.MinusCheckNext AND "A03_HMI".MB3.Button.A0302.Bordatrice.Regolazione.Passaggio_Combo[2].Bwd_Minus) OR ("A0302_Bordatrice_RegolazioneFormato".AX_M[4].COut.PlusCheckNext AND "A0302_Bordatrice_RegolazioneFormato".AX_M[5].COut.PlusCheckNext AND "A03_HMI".MB3.Button.A0302.Bordatrice.Regolazione.Passaggio_Combo[2].Fwd_Plus)) THEN
       #MB3_Decoder.OpEnabled := TRUE;
   END_IF;
   IF #_w1 AND NOT "A0302_Bordatrice_RegolazioneFormato".AX_M[4].COut.Standstill AND NOT "A0302_Bordatrice_RegolazioneFormato".AX_M[5].COut.Standstill THEN
       #MB3_Decoder.OpRunning := TRUE;
   END_IF;
   IF #_w1 AND (("A03_HMI".MB3.Button.A0302.Bordatrice.Regolazione.Passaggio_Combo[2].Bwd_Minus AND "A0302_Bordatrice_RegolazioneFormato".AX_M[4].COut.MinusLimitReached AND "A0302_Bordatrice_RegolazioneFormato".AX_M[5].COut.MinusLimitReached) OR ("A03_HMI".MB3.Button.A0302.Bordatrice.Regolazione.Passaggio_Combo[2].Fwd_Plus AND "A0302_Bordatrice_RegolazioneFormato".AX_M[4].COut.PlusLimitReached AND "A0302_Bordatrice_RegolazioneFormato".AX_M[5].COut.PlusLimitReached)) THEN
       #MB3_Decoder.OpDone := TRUE;
   END_IF;
END_REGION

REGION Network 41: MB3 Code 4089 - REGOLAZ. BORDATRICE - PASSAGGIO 02 - COMBO AX-POS
   RUNG wire#powerrail
      { S7_Templates := "SrcType := Int" } EQ_Contact(in1 := #MB3_Decoder.Code, in2 := #"4089_BORDATRICE_PASS02-COMBO_AX-POS")
      wire#w1
      { S7_Templates := "SrcType := LReal" } NE_Contact(in1 := "A0302_Bordatrice_RegolazioneFormato".AX_M[4].COut.ActualPosition, in2 := "A0302_Bordatrice_RegolazioneFormato".HMI.Passaggio02_Combo_TargetPos)
      wire#w2
      Contact( #MB3_Decoder.OperationPlus )
      Coil( "A03_HMI".MB3.Button.A0302.Bordatrice.Regolazione.Passaggio_Combo[2].MoveToPos )
   END_RUNG
   RUNG wire#w1
      { S7_Templates := "SrcType := LReal" } NE_Contact(in1 := "A0302_Bordatrice_RegolazioneFormato".AX_M[5].COut.ActualPosition, in2 := "A0302_Bordatrice_RegolazioneFormato".HMI.Passaggio02_Combo_TargetPos)
   END_RUNG wire#w2
   RUNG wire#w1
      Contact( TRUE )
      S_Coil( #MB3_Decoder.OpEnabled )
   END_RUNG
   RUNG wire#w1
      I_Contact( "A0302_Bordatrice_RegolazioneFormato".AX_M[4].COut.Standstill )
      wire#w3
      S_Coil( #MB3_Decoder.OpRunning )
   END_RUNG
   RUNG wire#w1
      I_Contact( "A0302_Bordatrice_RegolazioneFormato".AX_M[5].COut.Standstill )
   END_RUNG wire#w3
   RUNG wire#w1
      Contact( "A0302_Bordatrice_RegolazioneFormato".AX_M[4].COut.InPosition )
      Contact( "A0302_Bordatrice_RegolazioneFormato".AX_M[5].COut.InPosition )
      S_Coil( #MB3_Decoder.OpDone )
   END_RUNG
   // the same network as SCL:
   #_w1 := #MB3_Decoder.Code = #"4089_BORDATRICE_PASS02-COMBO_AX-POS";
   "A03_HMI".MB3.Button.A0302.Bordatrice.Regolazione.Passaggio_Combo[2].MoveToPos := #_w1 AND (("A0302_Bordatrice_RegolazioneFormato".AX_M[4].COut.ActualPosition <> "A0302_Bordatrice_RegolazioneFormato".HMI.Passaggio02_Combo_TargetPos) OR ("A0302_Bordatrice_RegolazioneFormato".AX_M[5].COut.ActualPosition <> "A0302_Bordatrice_RegolazioneFormato".HMI.Passaggio02_Combo_TargetPos)) AND #MB3_Decoder.OperationPlus;
   IF #_w1 AND TRUE THEN #MB3_Decoder.OpEnabled := TRUE; END_IF;
   IF #_w1 AND (NOT "A0302_Bordatrice_RegolazioneFormato".AX_M[4].COut.Standstill OR NOT "A0302_Bordatrice_RegolazioneFormato".AX_M[5].COut.Standstill) THEN
       #MB3_Decoder.OpRunning := TRUE;
   END_IF;
   IF #_w1 AND "A0302_Bordatrice_RegolazioneFormato".AX_M[4].COut.InPosition AND "A0302_Bordatrice_RegolazioneFormato".AX_M[5].COut.InPosition THEN
       #MB3_Decoder.OpDone := TRUE;
   END_IF;
END_REGION

REGION Network 42: MB3 Code 4082 - REGOLAZ. BORDATRICE - PASSAGGIO 02 - LATO-OP
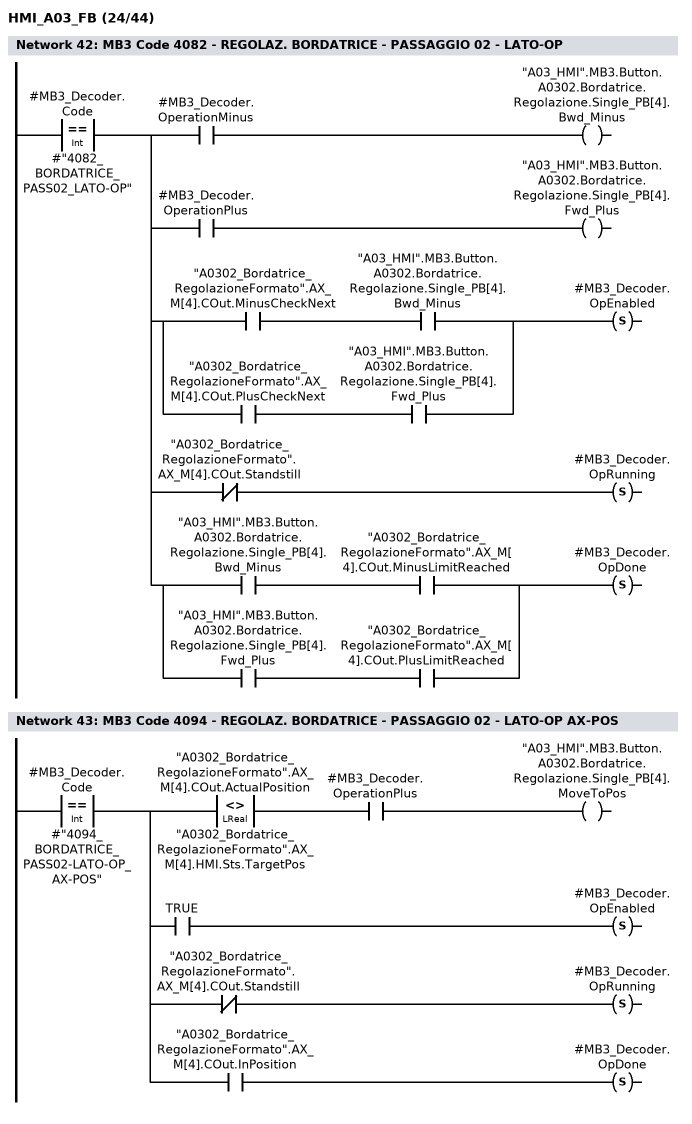
   RUNG wire#powerrail
      { S7_Templates := "SrcType := Int" } EQ_Contact(in1 := #MB3_Decoder.Code, in2 := #"4082_BORDATRICE_PASS02_LATO-OP")
      wire#w1
      Contact( #MB3_Decoder.OperationMinus )
      Coil( "A03_HMI".MB3.Button.A0302.Bordatrice.Regolazione.Single_PB[4].Bwd_Minus )
   END_RUNG
   RUNG wire#w1
      Contact( #MB3_Decoder.OperationPlus )
      Coil( "A03_HMI".MB3.Button.A0302.Bordatrice.Regolazione.Single_PB[4].Fwd_Plus )
   END_RUNG
   RUNG wire#w1
      Contact( "A0302_Bordatrice_RegolazioneFormato".AX_M[4].COut.MinusCheckNext )
      Contact( "A03_HMI".MB3.Button.A0302.Bordatrice.Regolazione.Single_PB[4].Bwd_Minus )
      wire#w2
      S_Coil( #MB3_Decoder.OpEnabled )
   END_RUNG
   RUNG wire#w1
      Contact( "A0302_Bordatrice_RegolazioneFormato".AX_M[4].COut.PlusCheckNext )
      Contact( "A03_HMI".MB3.Button.A0302.Bordatrice.Regolazione.Single_PB[4].Fwd_Plus )
   END_RUNG wire#w2
   RUNG wire#w1
      I_Contact( "A0302_Bordatrice_RegolazioneFormato".AX_M[4].COut.Standstill )
      S_Coil( #MB3_Decoder.OpRunning )
   END_RUNG
   RUNG wire#w1
      Contact( "A03_HMI".MB3.Button.A0302.Bordatrice.Regolazione.Single_PB[4].Bwd_Minus )
      Contact( "A0302_Bordatrice_RegolazioneFormato".AX_M[4].COut.MinusLimitReached )
      wire#w3
      S_Coil( #MB3_Decoder.OpDone )
   END_RUNG
   RUNG wire#w1
      Contact( "A03_HMI".MB3.Button.A0302.Bordatrice.Regolazione.Single_PB[4].Fwd_Plus )
      Contact( "A0302_Bordatrice_RegolazioneFormato".AX_M[4].COut.PlusLimitReached )
   END_RUNG wire#w3
   // the same network as SCL:
   #_w1 := #MB3_Decoder.Code = #"4082_BORDATRICE_PASS02_LATO-OP";
   "A03_HMI".MB3.Button.A0302.Bordatrice.Regolazione.Single_PB[4].Bwd_Minus := #_w1 AND #MB3_Decoder.OperationMinus;
   "A03_HMI".MB3.Button.A0302.Bordatrice.Regolazione.Single_PB[4].Fwd_Plus := #_w1 AND #MB3_Decoder.OperationPlus;
   IF #_w1 AND (("A0302_Bordatrice_RegolazioneFormato".AX_M[4].COut.MinusCheckNext AND "A03_HMI".MB3.Button.A0302.Bordatrice.Regolazione.Single_PB[4].Bwd_Minus) OR ("A0302_Bordatrice_RegolazioneFormato".AX_M[4].COut.PlusCheckNext AND "A03_HMI".MB3.Button.A0302.Bordatrice.Regolazione.Single_PB[4].Fwd_Plus)) THEN
       #MB3_Decoder.OpEnabled := TRUE;
   END_IF;
   IF #_w1 AND NOT "A0302_Bordatrice_RegolazioneFormato".AX_M[4].COut.Standstill THEN
       #MB3_Decoder.OpRunning := TRUE;
   END_IF;
   IF #_w1 AND (("A03_HMI".MB3.Button.A0302.Bordatrice.Regolazione.Single_PB[4].Bwd_Minus AND "A0302_Bordatrice_RegolazioneFormato".AX_M[4].COut.MinusLimitReached) OR ("A03_HMI".MB3.Button.A0302.Bordatrice.Regolazione.Single_PB[4].Fwd_Plus AND "A0302_Bordatrice_RegolazioneFormato".AX_M[4].COut.PlusLimitReached)) THEN
       #MB3_Decoder.OpDone := TRUE;
   END_IF;
END_REGION

REGION Network 43: MB3 Code 4094 - REGOLAZ. BORDATRICE - PASSAGGIO 02 - LATO-OP AX-POS
   RUNG wire#powerrail
      { S7_Templates := "SrcType := Int" } EQ_Contact(in1 := #MB3_Decoder.Code, in2 := #"4094_BORDATRICE_PASS02-LATO-OP_AX-POS")
      wire#w1
      { S7_Templates := "SrcType := LReal" } NE_Contact(in1 := "A0302_Bordatrice_RegolazioneFormato".AX_M[4].COut.ActualPosition, in2 := "A0302_Bordatrice_RegolazioneFormato".AX_M[4].HMI.Sts.TargetPos)
      Contact( #MB3_Decoder.OperationPlus )
      Coil( "A03_HMI".MB3.Button.A0302.Bordatrice.Regolazione.Single_PB[4].MoveToPos )
   END_RUNG
   RUNG wire#w1
      Contact( TRUE )
      S_Coil( #MB3_Decoder.OpEnabled )
   END_RUNG
   RUNG wire#w1
      I_Contact( "A0302_Bordatrice_RegolazioneFormato".AX_M[4].COut.Standstill )
      S_Coil( #MB3_Decoder.OpRunning )
   END_RUNG
   RUNG wire#w1
      Contact( "A0302_Bordatrice_RegolazioneFormato".AX_M[4].COut.InPosition )
      S_Coil( #MB3_Decoder.OpDone )
   END_RUNG
   // the same network as SCL:
   #_w1 := #MB3_Decoder.Code = #"4094_BORDATRICE_PASS02-LATO-OP_AX-POS";
   "A03_HMI".MB3.Button.A0302.Bordatrice.Regolazione.Single_PB[4].MoveToPos := #_w1 AND ("A0302_Bordatrice_RegolazioneFormato".AX_M[4].COut.ActualPosition <> "A0302_Bordatrice_RegolazioneFormato".AX_M[4].HMI.Sts.TargetPos) AND #MB3_Decoder.OperationPlus;
   IF #_w1 AND TRUE THEN #MB3_Decoder.OpEnabled := TRUE; END_IF;
   IF #_w1 AND NOT "A0302_Bordatrice_RegolazioneFormato".AX_M[4].COut.Standstill THEN
       #MB3_Decoder.OpRunning := TRUE;
   END_IF;
   IF #_w1 AND "A0302_Bordatrice_RegolazioneFormato".AX_M[4].COut.InPosition THEN
       #MB3_Decoder.OpDone := TRUE;
   END_IF;
END_REGION

REGION Network 44: MB3 Code 4083 - REGOLAZ. BORDATRICE - PASSAGGIO 02 - LATO-MOT
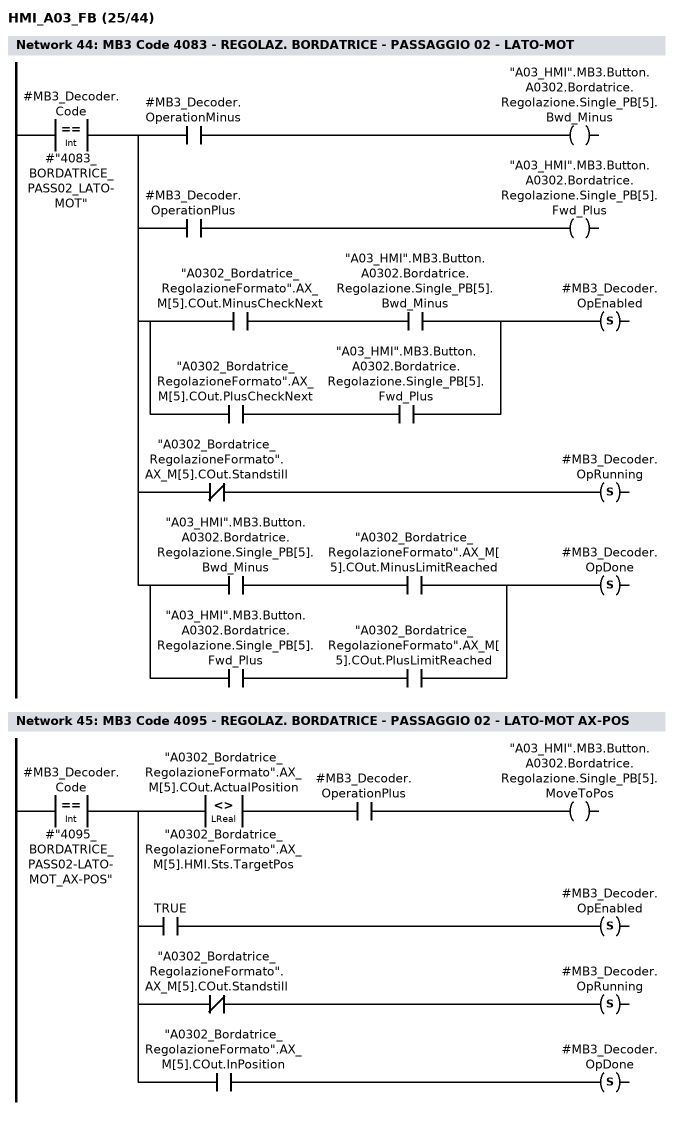
   RUNG wire#powerrail
      { S7_Templates := "SrcType := Int" } EQ_Contact(in1 := #MB3_Decoder.Code, in2 := #"4083_BORDATRICE_PASS02_LATO-MOT")
      wire#w1
      Contact( #MB3_Decoder.OperationMinus )
      Coil( "A03_HMI".MB3.Button.A0302.Bordatrice.Regolazione.Single_PB[5].Bwd_Minus )
   END_RUNG
   RUNG wire#w1
      Contact( #MB3_Decoder.OperationPlus )
      Coil( "A03_HMI".MB3.Button.A0302.Bordatrice.Regolazione.Single_PB[5].Fwd_Plus )
   END_RUNG
   RUNG wire#w1
      Contact( "A0302_Bordatrice_RegolazioneFormato".AX_M[5].COut.MinusCheckNext )
      Contact( "A03_HMI".MB3.Button.A0302.Bordatrice.Regolazione.Single_PB[5].Bwd_Minus )
      wire#w2
      S_Coil( #MB3_Decoder.OpEnabled )
   END_RUNG
   RUNG wire#w1
      Contact( "A0302_Bordatrice_RegolazioneFormato".AX_M[5].COut.PlusCheckNext )
      Contact( "A03_HMI".MB3.Button.A0302.Bordatrice.Regolazione.Single_PB[5].Fwd_Plus )
   END_RUNG wire#w2
   RUNG wire#w1
      I_Contact( "A0302_Bordatrice_RegolazioneFormato".AX_M[5].COut.Standstill )
      S_Coil( #MB3_Decoder.OpRunning )
   END_RUNG
   RUNG wire#w1
      Contact( "A03_HMI".MB3.Button.A0302.Bordatrice.Regolazione.Single_PB[5].Bwd_Minus )
      Contact( "A0302_Bordatrice_RegolazioneFormato".AX_M[5].COut.MinusLimitReached )
      wire#w3
      S_Coil( #MB3_Decoder.OpDone )
   END_RUNG
   RUNG wire#w1
      Contact( "A03_HMI".MB3.Button.A0302.Bordatrice.Regolazione.Single_PB[5].Fwd_Plus )
      Contact( "A0302_Bordatrice_RegolazioneFormato".AX_M[5].COut.PlusLimitReached )
   END_RUNG wire#w3
   // the same network as SCL:
   #_w1 := #MB3_Decoder.Code = #"4083_BORDATRICE_PASS02_LATO-MOT";
   "A03_HMI".MB3.Button.A0302.Bordatrice.Regolazione.Single_PB[5].Bwd_Minus := #_w1 AND #MB3_Decoder.OperationMinus;
   "A03_HMI".MB3.Button.A0302.Bordatrice.Regolazione.Single_PB[5].Fwd_Plus := #_w1 AND #MB3_Decoder.OperationPlus;
   IF #_w1 AND (("A0302_Bordatrice_RegolazioneFormato".AX_M[5].COut.MinusCheckNext AND "A03_HMI".MB3.Button.A0302.Bordatrice.Regolazione.Single_PB[5].Bwd_Minus) OR ("A0302_Bordatrice_RegolazioneFormato".AX_M[5].COut.PlusCheckNext AND "A03_HMI".MB3.Button.A0302.Bordatrice.Regolazione.Single_PB[5].Fwd_Plus)) THEN
       #MB3_Decoder.OpEnabled := TRUE;
   END_IF;
   IF #_w1 AND NOT "A0302_Bordatrice_RegolazioneFormato".AX_M[5].COut.Standstill THEN
       #MB3_Decoder.OpRunning := TRUE;
   END_IF;
   IF #_w1 AND (("A03_HMI".MB3.Button.A0302.Bordatrice.Regolazione.Single_PB[5].Bwd_Minus AND "A0302_Bordatrice_RegolazioneFormato".AX_M[5].COut.MinusLimitReached) OR ("A03_HMI".MB3.Button.A0302.Bordatrice.Regolazione.Single_PB[5].Fwd_Plus AND "A0302_Bordatrice_RegolazioneFormato".AX_M[5].COut.PlusLimitReached)) THEN
       #MB3_Decoder.OpDone := TRUE;
   END_IF;
END_REGION

REGION Network 45: MB3 Code 4095 - REGOLAZ. BORDATRICE - PASSAGGIO 02 - LATO-MOT AX-POS
   RUNG wire#powerrail
      { S7_Templates := "SrcType := Int" } EQ_Contact(in1 := #MB3_Decoder.Code, in2 := #"4095_BORDATRICE_PASS02-LATO-MOT_AX-POS")
      wire#w1
      { S7_Templates := "SrcType := LReal" } NE_Contact(in1 := "A0302_Bordatrice_RegolazioneFormato".AX_M[5].COut.ActualPosition, in2 := "A0302_Bordatrice_RegolazioneFormato".AX_M[5].HMI.Sts.TargetPos)
      Contact( #MB3_Decoder.OperationPlus )
      Coil( "A03_HMI".MB3.Button.A0302.Bordatrice.Regolazione.Single_PB[5].MoveToPos )
   END_RUNG
   RUNG wire#w1
      Contact( TRUE )
      S_Coil( #MB3_Decoder.OpEnabled )
   END_RUNG
   RUNG wire#w1
      I_Contact( "A0302_Bordatrice_RegolazioneFormato".AX_M[5].COut.Standstill )
      S_Coil( #MB3_Decoder.OpRunning )
   END_RUNG
   RUNG wire#w1
      Contact( "A0302_Bordatrice_RegolazioneFormato".AX_M[5].COut.InPosition )
      S_Coil( #MB3_Decoder.OpDone )
   END_RUNG
   // the same network as SCL:
   #_w1 := #MB3_Decoder.Code = #"4095_BORDATRICE_PASS02-LATO-MOT_AX-POS";
   "A03_HMI".MB3.Button.A0302.Bordatrice.Regolazione.Single_PB[5].MoveToPos := #_w1 AND ("A0302_Bordatrice_RegolazioneFormato".AX_M[5].COut.ActualPosition <> "A0302_Bordatrice_RegolazioneFormato".AX_M[5].HMI.Sts.TargetPos) AND #MB3_Decoder.OperationPlus;
   IF #_w1 AND TRUE THEN #MB3_Decoder.OpEnabled := TRUE; END_IF;
   IF #_w1 AND NOT "A0302_Bordatrice_RegolazioneFormato".AX_M[5].COut.Standstill THEN
       #MB3_Decoder.OpRunning := TRUE;
   END_IF;
   IF #_w1 AND "A0302_Bordatrice_RegolazioneFormato".AX_M[5].COut.InPosition THEN
       #MB3_Decoder.OpDone := TRUE;
   END_IF;
END_REGION

REGION Network 46: MB3 Code 4036 - REGOLAZ. BORDATRICE - PASSAGGIO 03 - COMBO
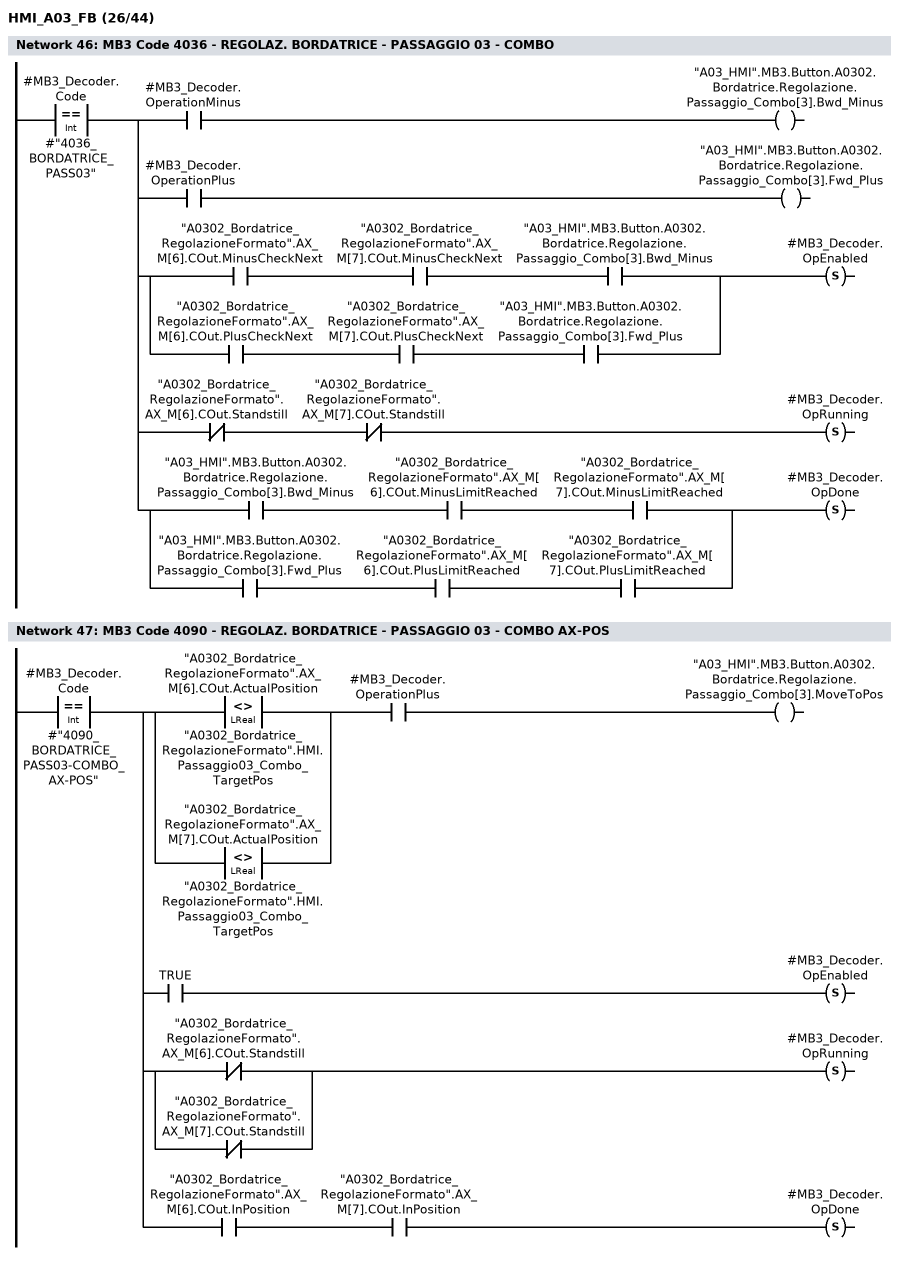
   RUNG wire#powerrail
      { S7_Templates := "SrcType := Int" } EQ_Contact(in1 := #MB3_Decoder.Code, in2 := #"4036_BORDATRICE_PASS03")
      wire#w1
      Contact( #MB3_Decoder.OperationMinus )
      Coil( "A03_HMI".MB3.Button.A0302.Bordatrice.Regolazione.Passaggio_Combo[3].Bwd_Minus )
   END_RUNG
   RUNG wire#w1
      Contact( #MB3_Decoder.OperationPlus )
      Coil( "A03_HMI".MB3.Button.A0302.Bordatrice.Regolazione.Passaggio_Combo[3].Fwd_Plus )
   END_RUNG
   RUNG wire#w1
      Contact( "A0302_Bordatrice_RegolazioneFormato".AX_M[6].COut.MinusCheckNext )
      Contact( "A0302_Bordatrice_RegolazioneFormato".AX_M[7].COut.MinusCheckNext )
      Contact( "A03_HMI".MB3.Button.A0302.Bordatrice.Regolazione.Passaggio_Combo[3].Bwd_Minus )
      wire#w2
      S_Coil( #MB3_Decoder.OpEnabled )
   END_RUNG
   RUNG wire#w1
      Contact( "A0302_Bordatrice_RegolazioneFormato".AX_M[6].COut.PlusCheckNext )
      Contact( "A0302_Bordatrice_RegolazioneFormato".AX_M[7].COut.PlusCheckNext )
      Contact( "A03_HMI".MB3.Button.A0302.Bordatrice.Regolazione.Passaggio_Combo[3].Fwd_Plus )
   END_RUNG wire#w2
   RUNG wire#w1
      I_Contact( "A0302_Bordatrice_RegolazioneFormato".AX_M[6].COut.Standstill )
      I_Contact( "A0302_Bordatrice_RegolazioneFormato".AX_M[7].COut.Standstill )
      S_Coil( #MB3_Decoder.OpRunning )
   END_RUNG
   RUNG wire#w1
      Contact( "A03_HMI".MB3.Button.A0302.Bordatrice.Regolazione.Passaggio_Combo[3].Bwd_Minus )
      Contact( "A0302_Bordatrice_RegolazioneFormato".AX_M[6].COut.MinusLimitReached )
      Contact( "A0302_Bordatrice_RegolazioneFormato".AX_M[7].COut.MinusLimitReached )
      wire#w3
      S_Coil( #MB3_Decoder.OpDone )
   END_RUNG
   RUNG wire#w1
      Contact( "A03_HMI".MB3.Button.A0302.Bordatrice.Regolazione.Passaggio_Combo[3].Fwd_Plus )
      Contact( "A0302_Bordatrice_RegolazioneFormato".AX_M[6].COut.PlusLimitReached )
      Contact( "A0302_Bordatrice_RegolazioneFormato".AX_M[7].COut.PlusLimitReached )
   END_RUNG wire#w3
   // the same network as SCL:
   #_w1 := #MB3_Decoder.Code = #"4036_BORDATRICE_PASS03";
   "A03_HMI".MB3.Button.A0302.Bordatrice.Regolazione.Passaggio_Combo[3].Bwd_Minus := #_w1 AND #MB3_Decoder.OperationMinus;
   "A03_HMI".MB3.Button.A0302.Bordatrice.Regolazione.Passaggio_Combo[3].Fwd_Plus := #_w1 AND #MB3_Decoder.OperationPlus;
   IF #_w1 AND (("A0302_Bordatrice_RegolazioneFormato".AX_M[6].COut.MinusCheckNext AND "A0302_Bordatrice_RegolazioneFormato".AX_M[7].COut.MinusCheckNext AND "A03_HMI".MB3.Button.A0302.Bordatrice.Regolazione.Passaggio_Combo[3].Bwd_Minus) OR ("A0302_Bordatrice_RegolazioneFormato".AX_M[6].COut.PlusCheckNext AND "A0302_Bordatrice_RegolazioneFormato".AX_M[7].COut.PlusCheckNext AND "A03_HMI".MB3.Button.A0302.Bordatrice.Regolazione.Passaggio_Combo[3].Fwd_Plus)) THEN
       #MB3_Decoder.OpEnabled := TRUE;
   END_IF;
   IF #_w1 AND NOT "A0302_Bordatrice_RegolazioneFormato".AX_M[6].COut.Standstill AND NOT "A0302_Bordatrice_RegolazioneFormato".AX_M[7].COut.Standstill THEN
       #MB3_Decoder.OpRunning := TRUE;
   END_IF;
   IF #_w1 AND (("A03_HMI".MB3.Button.A0302.Bordatrice.Regolazione.Passaggio_Combo[3].Bwd_Minus AND "A0302_Bordatrice_RegolazioneFormato".AX_M[6].COut.MinusLimitReached AND "A0302_Bordatrice_RegolazioneFormato".AX_M[7].COut.MinusLimitReached) OR ("A03_HMI".MB3.Button.A0302.Bordatrice.Regolazione.Passaggio_Combo[3].Fwd_Plus AND "A0302_Bordatrice_RegolazioneFormato".AX_M[6].COut.PlusLimitReached AND "A0302_Bordatrice_RegolazioneFormato".AX_M[7].COut.PlusLimitReached)) THEN
       #MB3_Decoder.OpDone := TRUE;
   END_IF;
END_REGION

REGION Network 47: MB3 Code 4090 - REGOLAZ. BORDATRICE - PASSAGGIO 03 - COMBO AX-POS
   RUNG wire#powerrail
      { S7_Templates := "SrcType := Int" } EQ_Contact(in1 := #MB3_Decoder.Code, in2 := #"4090_BORDATRICE_PASS03-COMBO_AX-POS")
      wire#w1
      { S7_Templates := "SrcType := LReal" } NE_Contact(in1 := "A0302_Bordatrice_RegolazioneFormato".AX_M[6].COut.ActualPosition, in2 := "A0302_Bordatrice_RegolazioneFormato".HMI.Passaggio03_Combo_TargetPos)
      wire#w2
      Contact( #MB3_Decoder.OperationPlus )
      Coil( "A03_HMI".MB3.Button.A0302.Bordatrice.Regolazione.Passaggio_Combo[3].MoveToPos )
   END_RUNG
   RUNG wire#w1
      { S7_Templates := "SrcType := LReal" } NE_Contact(in1 := "A0302_Bordatrice_RegolazioneFormato".AX_M[7].COut.ActualPosition, in2 := "A0302_Bordatrice_RegolazioneFormato".HMI.Passaggio03_Combo_TargetPos)
   END_RUNG wire#w2
   RUNG wire#w1
      Contact( TRUE )
      S_Coil( #MB3_Decoder.OpEnabled )
   END_RUNG
   RUNG wire#w1
      I_Contact( "A0302_Bordatrice_RegolazioneFormato".AX_M[6].COut.Standstill )
      wire#w3
      S_Coil( #MB3_Decoder.OpRunning )
   END_RUNG
   RUNG wire#w1
      I_Contact( "A0302_Bordatrice_RegolazioneFormato".AX_M[7].COut.Standstill )
   END_RUNG wire#w3
   RUNG wire#w1
      Contact( "A0302_Bordatrice_RegolazioneFormato".AX_M[6].COut.InPosition )
      Contact( "A0302_Bordatrice_RegolazioneFormato".AX_M[7].COut.InPosition )
      S_Coil( #MB3_Decoder.OpDone )
   END_RUNG
   // the same network as SCL:
   #_w1 := #MB3_Decoder.Code = #"4090_BORDATRICE_PASS03-COMBO_AX-POS";
   "A03_HMI".MB3.Button.A0302.Bordatrice.Regolazione.Passaggio_Combo[3].MoveToPos := #_w1 AND (("A0302_Bordatrice_RegolazioneFormato".AX_M[6].COut.ActualPosition <> "A0302_Bordatrice_RegolazioneFormato".HMI.Passaggio03_Combo_TargetPos) OR ("A0302_Bordatrice_RegolazioneFormato".AX_M[7].COut.ActualPosition <> "A0302_Bordatrice_RegolazioneFormato".HMI.Passaggio03_Combo_TargetPos)) AND #MB3_Decoder.OperationPlus;
   IF #_w1 AND TRUE THEN #MB3_Decoder.OpEnabled := TRUE; END_IF;
   IF #_w1 AND (NOT "A0302_Bordatrice_RegolazioneFormato".AX_M[6].COut.Standstill OR NOT "A0302_Bordatrice_RegolazioneFormato".AX_M[7].COut.Standstill) THEN
       #MB3_Decoder.OpRunning := TRUE;
   END_IF;
   IF #_w1 AND "A0302_Bordatrice_RegolazioneFormato".AX_M[6].COut.InPosition AND "A0302_Bordatrice_RegolazioneFormato".AX_M[7].COut.InPosition THEN
       #MB3_Decoder.OpDone := TRUE;
   END_IF;
END_REGION

REGION Network 48: MB3 Code 4084 - REGOLAZ. BORDATRICE - PASSAGGIO 03 - LATO-OP
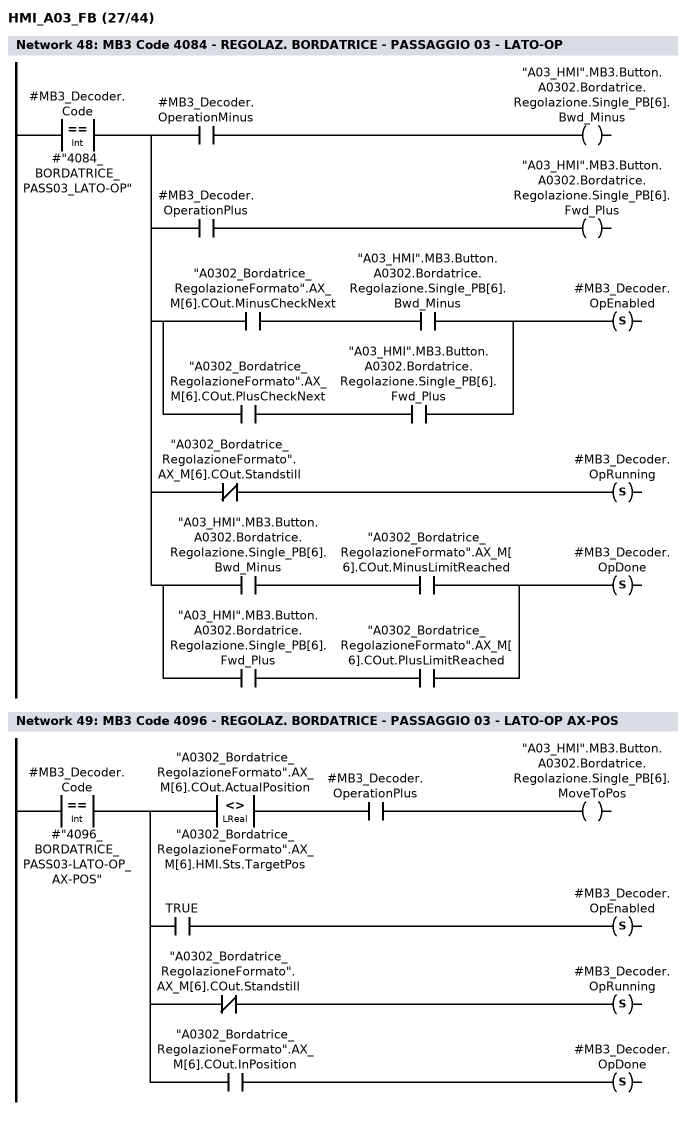
   RUNG wire#powerrail
      { S7_Templates := "SrcType := Int" } EQ_Contact(in1 := #MB3_Decoder.Code, in2 := #"4084_BORDATRICE_PASS03_LATO-OP")
      wire#w1
      Contact( #MB3_Decoder.OperationMinus )
      Coil( "A03_HMI".MB3.Button.A0302.Bordatrice.Regolazione.Single_PB[6].Bwd_Minus )
   END_RUNG
   RUNG wire#w1
      Contact( #MB3_Decoder.OperationPlus )
      Coil( "A03_HMI".MB3.Button.A0302.Bordatrice.Regolazione.Single_PB[6].Fwd_Plus )
   END_RUNG
   RUNG wire#w1
      Contact( "A0302_Bordatrice_RegolazioneFormato".AX_M[6].COut.MinusCheckNext )
      Contact( "A03_HMI".MB3.Button.A0302.Bordatrice.Regolazione.Single_PB[6].Bwd_Minus )
      wire#w2
      S_Coil( #MB3_Decoder.OpEnabled )
   END_RUNG
   RUNG wire#w1
      Contact( "A0302_Bordatrice_RegolazioneFormato".AX_M[6].COut.PlusCheckNext )
      Contact( "A03_HMI".MB3.Button.A0302.Bordatrice.Regolazione.Single_PB[6].Fwd_Plus )
   END_RUNG wire#w2
   RUNG wire#w1
      I_Contact( "A0302_Bordatrice_RegolazioneFormato".AX_M[6].COut.Standstill )
      S_Coil( #MB3_Decoder.OpRunning )
   END_RUNG
   RUNG wire#w1
      Contact( "A03_HMI".MB3.Button.A0302.Bordatrice.Regolazione.Single_PB[6].Bwd_Minus )
      Contact( "A0302_Bordatrice_RegolazioneFormato".AX_M[6].COut.MinusLimitReached )
      wire#w3
      S_Coil( #MB3_Decoder.OpDone )
   END_RUNG
   RUNG wire#w1
      Contact( "A03_HMI".MB3.Button.A0302.Bordatrice.Regolazione.Single_PB[6].Fwd_Plus )
      Contact( "A0302_Bordatrice_RegolazioneFormato".AX_M[6].COut.PlusLimitReached )
   END_RUNG wire#w3
   // the same network as SCL:
   #_w1 := #MB3_Decoder.Code = #"4084_BORDATRICE_PASS03_LATO-OP";
   "A03_HMI".MB3.Button.A0302.Bordatrice.Regolazione.Single_PB[6].Bwd_Minus := #_w1 AND #MB3_Decoder.OperationMinus;
   "A03_HMI".MB3.Button.A0302.Bordatrice.Regolazione.Single_PB[6].Fwd_Plus := #_w1 AND #MB3_Decoder.OperationPlus;
   IF #_w1 AND (("A0302_Bordatrice_RegolazioneFormato".AX_M[6].COut.MinusCheckNext AND "A03_HMI".MB3.Button.A0302.Bordatrice.Regolazione.Single_PB[6].Bwd_Minus) OR ("A0302_Bordatrice_RegolazioneFormato".AX_M[6].COut.PlusCheckNext AND "A03_HMI".MB3.Button.A0302.Bordatrice.Regolazione.Single_PB[6].Fwd_Plus)) THEN
       #MB3_Decoder.OpEnabled := TRUE;
   END_IF;
   IF #_w1 AND NOT "A0302_Bordatrice_RegolazioneFormato".AX_M[6].COut.Standstill THEN
       #MB3_Decoder.OpRunning := TRUE;
   END_IF;
   IF #_w1 AND (("A03_HMI".MB3.Button.A0302.Bordatrice.Regolazione.Single_PB[6].Bwd_Minus AND "A0302_Bordatrice_RegolazioneFormato".AX_M[6].COut.MinusLimitReached) OR ("A03_HMI".MB3.Button.A0302.Bordatrice.Regolazione.Single_PB[6].Fwd_Plus AND "A0302_Bordatrice_RegolazioneFormato".AX_M[6].COut.PlusLimitReached)) THEN
       #MB3_Decoder.OpDone := TRUE;
   END_IF;
END_REGION

REGION Network 49: MB3 Code 4096 - REGOLAZ. BORDATRICE - PASSAGGIO 03 - LATO-OP AX-POS
   RUNG wire#powerrail
      { S7_Templates := "SrcType := Int" } EQ_Contact(in1 := #MB3_Decoder.Code, in2 := #"4096_BORDATRICE_PASS03-LATO-OP_AX-POS")
      wire#w1
      { S7_Templates := "SrcType := LReal" } NE_Contact(in1 := "A0302_Bordatrice_RegolazioneFormato".AX_M[6].COut.ActualPosition, in2 := "A0302_Bordatrice_RegolazioneFormato".AX_M[6].HMI.Sts.TargetPos)
      Contact( #MB3_Decoder.OperationPlus )
      Coil( "A03_HMI".MB3.Button.A0302.Bordatrice.Regolazione.Single_PB[6].MoveToPos )
   END_RUNG
   RUNG wire#w1
      Contact( TRUE )
      S_Coil( #MB3_Decoder.OpEnabled )
   END_RUNG
   RUNG wire#w1
      I_Contact( "A0302_Bordatrice_RegolazioneFormato".AX_M[6].COut.Standstill )
      S_Coil( #MB3_Decoder.OpRunning )
   END_RUNG
   RUNG wire#w1
      Contact( "A0302_Bordatrice_RegolazioneFormato".AX_M[6].COut.InPosition )
      S_Coil( #MB3_Decoder.OpDone )
   END_RUNG
   // the same network as SCL:
   #_w1 := #MB3_Decoder.Code = #"4096_BORDATRICE_PASS03-LATO-OP_AX-POS";
   "A03_HMI".MB3.Button.A0302.Bordatrice.Regolazione.Single_PB[6].MoveToPos := #_w1 AND ("A0302_Bordatrice_RegolazioneFormato".AX_M[6].COut.ActualPosition <> "A0302_Bordatrice_RegolazioneFormato".AX_M[6].HMI.Sts.TargetPos) AND #MB3_Decoder.OperationPlus;
   IF #_w1 AND TRUE THEN #MB3_Decoder.OpEnabled := TRUE; END_IF;
   IF #_w1 AND NOT "A0302_Bordatrice_RegolazioneFormato".AX_M[6].COut.Standstill THEN
       #MB3_Decoder.OpRunning := TRUE;
   END_IF;
   IF #_w1 AND "A0302_Bordatrice_RegolazioneFormato".AX_M[6].COut.InPosition THEN
       #MB3_Decoder.OpDone := TRUE;
   END_IF;
END_REGION

REGION Network 50: MB3 Code 4085 - REGOLAZ. BORDATRICE - PASSAGGIO 03 - LATO-MOT
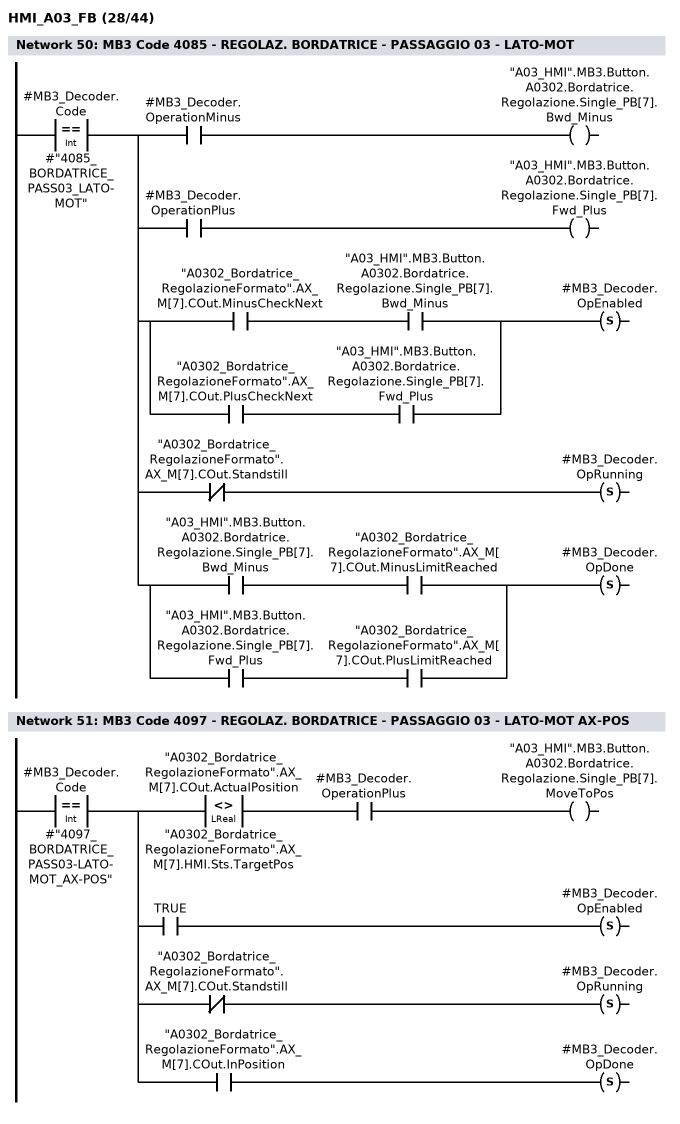
   RUNG wire#powerrail
      { S7_Templates := "SrcType := Int" } EQ_Contact(in1 := #MB3_Decoder.Code, in2 := #"4085_BORDATRICE_PASS03_LATO-MOT")
      wire#w1
      Contact( #MB3_Decoder.OperationMinus )
      Coil( "A03_HMI".MB3.Button.A0302.Bordatrice.Regolazione.Single_PB[7].Bwd_Minus )
   END_RUNG
   RUNG wire#w1
      Contact( #MB3_Decoder.OperationPlus )
      Coil( "A03_HMI".MB3.Button.A0302.Bordatrice.Regolazione.Single_PB[7].Fwd_Plus )
   END_RUNG
   RUNG wire#w1
      Contact( "A0302_Bordatrice_RegolazioneFormato".AX_M[7].COut.MinusCheckNext )
      Contact( "A03_HMI".MB3.Button.A0302.Bordatrice.Regolazione.Single_PB[7].Bwd_Minus )
      wire#w2
      S_Coil( #MB3_Decoder.OpEnabled )
   END_RUNG
   RUNG wire#w1
      Contact( "A0302_Bordatrice_RegolazioneFormato".AX_M[7].COut.PlusCheckNext )
      Contact( "A03_HMI".MB3.Button.A0302.Bordatrice.Regolazione.Single_PB[7].Fwd_Plus )
   END_RUNG wire#w2
   RUNG wire#w1
      I_Contact( "A0302_Bordatrice_RegolazioneFormato".AX_M[7].COut.Standstill )
      S_Coil( #MB3_Decoder.OpRunning )
   END_RUNG
   RUNG wire#w1
      Contact( "A03_HMI".MB3.Button.A0302.Bordatrice.Regolazione.Single_PB[7].Bwd_Minus )
      Contact( "A0302_Bordatrice_RegolazioneFormato".AX_M[7].COut.MinusLimitReached )
      wire#w3
      S_Coil( #MB3_Decoder.OpDone )
   END_RUNG
   RUNG wire#w1
      Contact( "A03_HMI".MB3.Button.A0302.Bordatrice.Regolazione.Single_PB[7].Fwd_Plus )
      Contact( "A0302_Bordatrice_RegolazioneFormato".AX_M[7].COut.PlusLimitReached )
   END_RUNG wire#w3
   // the same network as SCL:
   #_w1 := #MB3_Decoder.Code = #"4085_BORDATRICE_PASS03_LATO-MOT";
   "A03_HMI".MB3.Button.A0302.Bordatrice.Regolazione.Single_PB[7].Bwd_Minus := #_w1 AND #MB3_Decoder.OperationMinus;
   "A03_HMI".MB3.Button.A0302.Bordatrice.Regolazione.Single_PB[7].Fwd_Plus := #_w1 AND #MB3_Decoder.OperationPlus;
   IF #_w1 AND (("A0302_Bordatrice_RegolazioneFormato".AX_M[7].COut.MinusCheckNext AND "A03_HMI".MB3.Button.A0302.Bordatrice.Regolazione.Single_PB[7].Bwd_Minus) OR ("A0302_Bordatrice_RegolazioneFormato".AX_M[7].COut.PlusCheckNext AND "A03_HMI".MB3.Button.A0302.Bordatrice.Regolazione.Single_PB[7].Fwd_Plus)) THEN
       #MB3_Decoder.OpEnabled := TRUE;
   END_IF;
   IF #_w1 AND NOT "A0302_Bordatrice_RegolazioneFormato".AX_M[7].COut.Standstill THEN
       #MB3_Decoder.OpRunning := TRUE;
   END_IF;
   IF #_w1 AND (("A03_HMI".MB3.Button.A0302.Bordatrice.Regolazione.Single_PB[7].Bwd_Minus AND "A0302_Bordatrice_RegolazioneFormato".AX_M[7].COut.MinusLimitReached) OR ("A03_HMI".MB3.Button.A0302.Bordatrice.Regolazione.Single_PB[7].Fwd_Plus AND "A0302_Bordatrice_RegolazioneFormato".AX_M[7].COut.PlusLimitReached)) THEN
       #MB3_Decoder.OpDone := TRUE;
   END_IF;
END_REGION

REGION Network 51: MB3 Code 4097 - REGOLAZ. BORDATRICE - PASSAGGIO 03 - LATO-MOT AX-POS
   RUNG wire#powerrail
      { S7_Templates := "SrcType := Int" } EQ_Contact(in1 := #MB3_Decoder.Code, in2 := #"4097_BORDATRICE_PASS03-LATO-MOT_AX-POS")
      wire#w1
      { S7_Templates := "SrcType := LReal" } NE_Contact(in1 := "A0302_Bordatrice_RegolazioneFormato".AX_M[7].COut.ActualPosition, in2 := "A0302_Bordatrice_RegolazioneFormato".AX_M[7].HMI.Sts.TargetPos)
      Contact( #MB3_Decoder.OperationPlus )
      Coil( "A03_HMI".MB3.Button.A0302.Bordatrice.Regolazione.Single_PB[7].MoveToPos )
   END_RUNG
   RUNG wire#w1
      Contact( TRUE )
      S_Coil( #MB3_Decoder.OpEnabled )
   END_RUNG
   RUNG wire#w1
      I_Contact( "A0302_Bordatrice_RegolazioneFormato".AX_M[7].COut.Standstill )
      S_Coil( #MB3_Decoder.OpRunning )
   END_RUNG
   RUNG wire#w1
      Contact( "A0302_Bordatrice_RegolazioneFormato".AX_M[7].COut.InPosition )
      S_Coil( #MB3_Decoder.OpDone )
   END_RUNG
   // the same network as SCL:
   #_w1 := #MB3_Decoder.Code = #"4097_BORDATRICE_PASS03-LATO-MOT_AX-POS";
   "A03_HMI".MB3.Button.A0302.Bordatrice.Regolazione.Single_PB[7].MoveToPos := #_w1 AND ("A0302_Bordatrice_RegolazioneFormato".AX_M[7].COut.ActualPosition <> "A0302_Bordatrice_RegolazioneFormato".AX_M[7].HMI.Sts.TargetPos) AND #MB3_Decoder.OperationPlus;
   IF #_w1 AND TRUE THEN #MB3_Decoder.OpEnabled := TRUE; END_IF;
   IF #_w1 AND NOT "A0302_Bordatrice_RegolazioneFormato".AX_M[7].COut.Standstill THEN
       #MB3_Decoder.OpRunning := TRUE;
   END_IF;
   IF #_w1 AND "A0302_Bordatrice_RegolazioneFormato".AX_M[7].COut.InPosition THEN
       #MB3_Decoder.OpDone := TRUE;
   END_IF;
END_REGION

